Yaskawa INFORM job: OK_R2_O57-69(2)(90,0)_OK.JBI

/JOB
//NAME OK_R2_O57-69(2)(90,0)_OK
///FOLDERNAME X4
//POS
///NPOS 520,520,520,19,0,0
///TOOL 0
///POSTYPE PULSE
///PULSE
C00000=135424,72899,29147,3537,85342,-3792
C00001=134013,95021,61136,4029,77105,-4505
C00002=134047,101087,71818,4077,73656,-4607
C00003=134047,101216,72822,4088,73105,-4626
C00004=134047,101094,71866,4078,73630,-4609
C00005=133936,105187,77198,4137,72460,-4688
C00006=134047,101094,71866,4078,73630,-4609
C00007=133891,92563,58880,4064,77236,-4542
C00008=133627,85963,47659,4101,80754,-4516
C00009=133378,81291,43989,7801,81727,-8797
C00010=135556,84120,49328,8109,79955,-9206
C00011=135353,86004,57272,9537,76429,-10987
C00012=135353,86080,58384,9559,75792,-11036
C00013=135353,86004,57272,9537,76429,-10987
C00014=135153,91305,63913,9646,75106,-11159
C00015=135353,86004,57272,9537,76429,-10987
C00016=133639,82412,51163,9948,78523,-11411
C00017=132974,76709,41280,10049,81708,-11379
C00018=129415,64165,26444,10967,84795,-12306
C00019=98130,23251,42660,41088,49358,-30036
C00020=100023,30312,51600,41655,47069,-30160
C00021=100756,35138,59019,42789,45164,-30789
C00022=100756,36680,62008,43506,44389,-31244
C00023=100756,35138,59019,42789,45164,-30789
C00024=101219,36605,60555,42806,44807,-30721
C00025=100756,35138,59019,42789,45164,-30789
C00026=97195,22233,43091,41783,49188,-30648
C00027=75566,-7998,8685,42436,90764,-48719
C00028=92276,-23915,-5509,33057,78026,-45242
C00029=92276,-23145,-3597,33137,77364,-45439
C00030=92276,-23560,-4626,33093,77717,-45333
C00031=120131,-37031,-23614,-4680,71033,-34550
C00032=120131,-36585,-22326,-4696,70470,-34528
C00033=120989,-36588,-22328,-4847,70519,-34222
C00034=120131,-36585,-22326,-4696,70470,-34528
C00035=120131,-40902,-37029,-4549,77279,-34785
C00036=99101,-76935,-92016,31014,74911,-20401
C00037=52587,-144740,-101483,60524,64363,65274
C00038=46989,-65360,-59229,62781,73103,77672
C00039=56832,-65466,-56421,59287,64983,77772
C00040=57148,-65688,-55453,59188,64110,77279
C00041=55649,-62097,-53047,61106,66880,78547
C00042=57237,-59710,-51792,60669,66110,79037
C00043=56277,-61326,-53166,60831,66721,78866
C00044=55441,-62561,-53810,61057,67127,78609
C00045=56207,-63985,-54541,61032,66503,78630
C00046=55438,-62578,-53813,61060,67126,78606
C00047=51973,-62323,-54701,62406,69323,78001
C00048=48054,-62529,-57040,62601,72472,77896
C00049=29811,-70761,-60283,66780,94863,53671
C00050=30965,-22538,-31531,67696,97011,56857
C00051=55044,-42598,-44870,68563,88788,43678
C00052=56249,-45120,-46406,68472,87844,43687
C00053=57925,-45354,-44812,68371,86292,43442
C00054=57925,-45174,-43802,68390,86084,43215
C00055=57925,-45354,-44812,68371,86292,43442
C00056=59167,-45210,-44726,68282,85469,43617
C00057=57925,-45354,-44812,68371,86292,43442
C00058=55819,-44223,-45863,68504,88181,43684
C00059=44722,-31045,-43816,69927,97696,44632
C00060=43071,-26445,-40665,70170,98951,44614
C00061=137799,-47230,-78474,-21502,98719,52766
C00062=127020,6423,-39070,-7004,99714,51816
C00063=127020,5137,-37554,-6966,98131,51906
C00064=128416,4382,-35850,-7239,96821,52416
C00065=128416,3847,-35017,-7224,96041,52460
C00066=128416,4148,-35496,-7233,96488,52435
C00067=130041,4566,-35136,-7580,96617,52937
C00068=129924,4205,-34639,-7545,96120,52933
C00069=129457,4078,-34747,-7447,96082,52788
C00070=130190,4712,-35256,-7614,96778,52976
C00071=132441,34102,-13092,-8124,98426,53576
C00072=149392,-6912,-25974,-9982,75562,31317
C00073=149173,-488,-12666,-10148,70714,31647
C00074=149173,-326,-10897,-10208,69722,31733
C00075=149173,-394,-11578,-10184,70101,31701
C00076=148123,2416,-9216,-9823,69962,31333
C00077=149173,-394,-11578,-10184,70101,31701
C00078=152478,4885,-6741,-15795,72623,37698
C00079=151455,3828,-7649,-15488,72442,37350
C00080=152478,4560,-12614,-15554,75946,37261
C00081=146445,-24647,-43161,-13522,78564,34847
C00082=131494,-80468,-98534,-7816,92108,53678
C00083=52065,-14099,-27709,42253,108676,-27596
C00084=76671,-130461,-121705,35735,90710,-50834
C00085=94829,-93442,-100428,28991,96183,-47377
C00086=110716,-92055,-82664,19311,98038,-51285
C00087=114275,-93352,-80055,19461,95045,-50478
C00088=118122,-92212,-76367,19656,92534,-49497
C00089=118129,-91398,-74848,19645,92046,-49575
C00090=118122,-92212,-76367,19656,92534,-49497
C00091=119808,-92271,-76389,19753,92113,-48959
C00092=118122,-92212,-76367,19656,92534,-49497
C00093=114499,-91094,-78376,19482,95112,-50387
C00094=110992,-89821,-80983,19339,98080,-51178
C00095=124454,-89651,-86550,-11137,94998,69701
C00096=122569,-92184,-83910,-11067,91866,69331
C00097=120652,-93960,-80852,-11027,88857,68936
C00098=120652,-93520,-79457,-11027,88237,68992
C00099=120652,-93960,-80852,-11027,88857,68936
C00100=120650,-97396,-81866,-11026,87737,69033
C00101=120652,-93960,-80852,-11027,88857,68936
C00102=118161,-93768,-80427,-10994,88357,68121
C00103=120652,-93960,-80852,-11027,88857,68936
C00104=120037,-91891,-82714,-11032,90945,68539
C00105=121981,-89592,-85452,-11099,94026,68936
C00106=122005,-89480,-97857,-11363,101580,68254
C00107=122005,-89427,-98101,-11372,101754,68238
C00108=119094,-95812,-115555,4544,90851,20867
C00109=116502,-111480,-109655,18779,62868,-21987
C00110=119472,-101923,-104261,17094,63743,-20698
C00111=121534,-96097,-100090,16016,63743,-19914
C00112=121534,-96194,-98882,16123,62979,-20025
C00113=112336,-84014,-94514,26506,72534,-27449
C00114=114298,-84401,-94682,25743,71847,-26864
C00115=121534,-96097,-100090,16016,63743,-19914
C00116=121514,-92242,-98700,15883,64832,-19765
C00117=121534,-96097,-100090,16016,63743,-19914
C00118=119823,-101836,-103002,17025,62972,-20682
C00119=116876,-111303,-108368,18711,62117,-21969
C00120=126032,-109701,-108999,-21760,66785,27050
C00121=122513,-101468,-103921,-20079,66940,25677
C00122=121483,-94377,-99419,-19507,67520,25186
C00123=121483,-94509,-98158,-19621,66724,25324
C00124=121483,-94377,-99419,-19507,67520,25186
C00125=119206,-94355,-99408,-18489,67008,24418
C00126=121483,-94377,-99419,-19507,67520,25186
C00127=121468,-91005,-98354,-19362,68535,25006
C00128=121483,-94377,-99419,-19507,67520,25186
C00129=124810,-108862,-107603,-21303,66070,26716
C00130=126981,-112864,-109311,-24940,61360,29729
C00131=123200,-104180,-104415,-22777,61614,28126
C00132=121230,-90686,-98732,-21152,64298,26805
C00133=121230,-90968,-97120,-21351,63235,27013
C00134=121230,-90806,-98119,-21226,63888,26884
C00135=118688,-90754,-98099,-19926,63280,26013
C00136=121230,-90721,-98563,-21173,64184,26826
C00137=121211,-84894,-96124,-20922,65577,26553
C00138=121230,-90686,-98732,-21152,64298,26805
C00139=121413,-93580,-100796,-21282,64141,26906
C00140=124847,-101623,-105736,-23178,64029,28268
C00141=120616,-95755,-103879,-23668,64726,45447
C00142=120621,-89459,-99052,-23623,64971,45396
C00143=103351,-79665,-99305,-783,71297,41010
C00144=120614,-97387,-102466,-23992,63157,45792
C00145=122354,-96256,-100860,-24938,63287,46459
C00146=100033,-102933,-105835,1367,63570,39915
C00147=94055,-138721,-112948,5183,49813,37109
C00148=86627,-164185,-115821,11591,39368,32593
C00149=96470,-180165,-126119,4784,36529,37522
C00150=120616,-95173,-105764,-23303,89544,42444
C00151=107191,-96001,-89285,-21702,28532,58770
C00152=107187,-93630,-79997,-25295,24388,60561
C00153=107188,-92928,-77886,-26213,23539,61010
C00154=112799,-77365,-77001,-28703,40381,63534
C00155=107081,-94020,-78768,-26067,23489,60939
C00156=108911,-93070,-77209,-29349,23678,62538
C00157=100995,-91828,-91259,-7616,48178,54187
C00158=103021,-103152,-96284,-14725,52035,64235
C00159=107822,-73722,-90278,-18203,77746,63273
C00160=110657,-50226,-86705,-20295,96355,61815
C00161=107202,-93991,-108886,-21178,109925,43661
C00162=120660,-73953,-111348,-177,99224,-835
C00163=120616,-96234,-101081,23944,56754,-46777
C00164=120615,-96493,-97034,24670,54353,-47364
C00165=120614,-96447,-94923,25055,53191,-47662
C00166=125103,-63544,-87949,17256,75790,-41512
C00167=118876,-96360,-94049,26267,53277,-48431
C00168=120612,-97621,-95709,25094,53083,-47691
C00169=123782,-105215,-109377,22364,82684,-38148
C00170=123367,-104493,-108204,22899,85714,-42144
C00171=120617,-94319,-107453,23464,90858,-42123
C00172=120617,-92878,-109780,23521,92858,-41729
C00173=120619,-86141,-115603,23930,99335,-40429
C00174=120619,-89012,-115558,-8782,73464,-77384
C00175=120618,-92353,-112869,-8941,70132,-77138
C00176=120618,-93422,-111698,-9011,68877,-77043
C00177=120616,-94109,-113157,-8979,69414,-77085
C00178=120318,-89311,-110489,-8778,70198,-77244
C00179=120618,-93688,-111329,-9132,68044,-76969
C00180=120618,-93957,-110924,-9216,67187,-76884
C00181=120618,-94299,-110440,-9161,65769,-76809
C00182=120618,-94831,-109599,-8469,63241,-76696
C00183=120617,-95145,-109027,-7071,61401,-76664
C00184=120617,-95217,-108863,-5672,60665,-76701
C00185=120618,-93036,-111930,-4923,63538,-76718
C00186=120618,-92960,-112001,-4009,63579,-76743
C00187=120618,-92691,-112274,-2433,64167,-76800
C00188=120618,-92166,-112798,-840,65602,-76863
C00189=120618,-91419,-113490,342,67708,-76910
C00190=120619,-90739,-114068,878,69589,-76936
C00191=120619,-89701,-115007,939,71612,-76812
C00192=120619,-88814,-115609,873,73870,-76855
C00193=120619,-87740,-116270,151,76574,-76959
C00194=120619,-86987,-116700,-1182,78540,-77121
C00195=120619,-86782,-116823,-2462,79296,-77267
C00196=120619,-90672,-114378,-3278,75949,-77117
C00197=120619,-90769,-114313,-4130,75889,-77177
C00198=120619,-91109,-114056,-5597,75252,-77256
C00199=120618,-91719,-113544,-7101,73764,-77286
C00200=120618,-92472,-112836,-8259,71637,-77242
C00201=120618,-92872,-112418,-8666,70405,-77193
C00202=120618,-93168,-112034,-8862,69621,-77111
C00203=120618,-93422,-111698,-9011,68877,-77043
C00204=120618,-92353,-112869,-8941,70132,-77138
C00205=120619,-89012,-115558,-8782,73464,-77384
C00206=120595,-119438,-127420,8829,91162,-8830
C00207=129025,-103888,-99333,-21372,86937,54976
C00208=120613,-94952,-86848,-20336,81911,52813
C00209=120613,-94069,-83278,-20415,80272,53091
C00210=106776,-118156,-87795,-9907,57184,33367
C00211=120519,-95091,-83551,-20421,79912,53118
C00212=122104,-92396,-81537,-20633,80446,53604
C00213=112247,-111724,-87315,-12944,66201,41339
C00214=120203,-93448,-81675,-16163,85448,56808
C00215=120729,-92509,-78586,-16225,84191,57156
C00216=121550,-94129,-79175,-15118,86186,61621
C00217=122418,-96212,-79737,-13214,89323,68733
C00218=120612,-93818,-82398,-13271,91824,67835
C00219=120613,-94827,-86367,-13308,93699,67633
C00220=120614,-96085,-95173,-13466,98348,67128
C00221=120625,-105302,-100360,-13404,96846,67297
C00222=102872,-120945,-93289,41313,52454,-35552
C00223=111052,-89986,-73102,36259,51528,-31574
C00224=114360,-89865,-71590,35102,49434,-30694
C00225=117526,-83033,-67896,32906,49195,-29120
C00226=113966,-89555,-70876,35431,49366,-30932
C00227=115650,-91167,-72721,34446,48930,-30213
C00228=116035,-87162,-73783,30522,57415,-33049
C00229=114870,-90750,-79036,28299,65889,-37708
C00230=114629,-93248,-83330,25887,75293,-43435
C00231=115086,-85156,-72081,25020,76812,-47005
C00232=114845,-96650,-75395,24460,77575,-52847
C00233=115266,-96292,-75579,23738,83016,-58597
C00234=112822,-91718,-77371,23458,91001,-62960
C00235=109330,-92095,-80656,23399,93677,-63722
C00236=110759,-94815,-97268,24043,101385,-61640
C00237=25230,-87703,-86789,41333,106155,71905
C00238=55862,19660,17206,68346,89547,53836
C00239=59225,37567,25812,69215,105770,42705
C00240=67658,42850,42597,68102,97125,40508
C00241=69496,40939,42743,68154,95469,40297
C00242=67599,42910,43858,67984,96867,40179
C00243=68366,42138,41747,68199,96713,40671
C00244=69496,40844,42642,68155,95474,40303
C00245=69202,26042,27763,68892,91580,41859
C00246=69430,8343,11443,69273,87154,43187
C00247=70515,-11168,-4593,69437,78895,44683
C00248=70497,-3239,1595,68550,83825,57162
C00249=68177,-4212,-1280,68454,85880,57398
C00250=65815,-3605,-3490,68417,88124,57797
C00251=46513,-27715,-22241,69125,80479,38621
C00252=7625,-19791,-74194,84461,116832,51132
C00253=98528,-26744,-48644,33463,55012,18344
C00254=113253,15209,27106,3834,50657,-3406
C00255=113409,21623,32322,3755,50736,-3338
C00256=112944,26693,40965,4138,48051,-3650
C00257=113472,24070,39362,3899,47665,-3430
C00258=113579,25546,39455,3805,48359,-3355
C00259=112978,26683,40955,4121,48050,-3635
C00260=112942,28151,43799,5754,47269,-5081
C00261=107858,34053,50994,19891,49698,-15260
C00262=107375,37871,55183,23682,51778,-19403
C00263=102416,58013,78822,34430,58031,-35011
C00264=101528,71839,96969,38749,59697,-40411
C00265=101833,70144,94845,38592,59915,-40184
C00266=99205,63215,84174,37575,62603,-39615
C00267=97180,56339,73463,36771,65900,-39269
C00268=108272,10166,23438,3323,45242,-19316
C00269=109103,10218,12469,2549,51979,-18742
C00270=102461,24196,25876,17974,57306,-30655
C00271=99785,30090,30578,21838,60128,-34061
C00272=99052,29053,30612,22206,59809,-34434
C00273=101478,26267,28203,21358,59216,-33547
C00274=98901,31355,34377,29186,63057,-41116
C00275=92009,66840,89116,42947,61850,-57046
C00276=89877,62120,80876,42077,64804,-56709
C00277=70258,15873,38394,48666,102593,-69187
C00278=68720,8010,42290,53616,94090,-68666
C00279=74407,27282,60534,55400,90233,-68095
C00280=74758,1474,21309,45746,90270,-65676
C00281=98607,12568,39814,-52966,86937,-78252
C00282=98596,22842,59344,-53301,82774,-75788
C00283=96296,21421,60413,-54092,80731,-75703
C00284=95348,20952,60953,-54433,79893,-75663
C00285=96117,19164,58324,-54129,80713,-75783
C00286=95662,23434,63388,-54370,79922,-75521
C00287=95503,21312,61702,-54422,79811,-75531
C00288=92574,18445,54645,-48983,79889,-68258
C00289=91800,17848,53101,-47601,79897,-67557
C00290=92530,17999,51917,-47342,80806,-67673
C00291=94302,18640,49262,-46764,83033,-67943
C00292=79003,18324,29303,-31626,94586,-4503
C00293=64136,40618,57122,-29721,84915,-83830
C00294=62802,39067,58740,-29997,82892,-83805
C00295=62255,38544,59506,-30121,82059,-83791
C00296=62254,37103,56589,-30066,82978,-84033
C00297=62821,40643,61741,-30049,81995,-83562
C00298=59984,48909,70165,-26795,84201,-83115
C00299=59410,69261,96131,-25367,86084,-74959
C00300=59404,69357,96256,-25356,86081,-74939
C00301=59713,70793,96681,-25260,86600,-74945
C00302=60461,74839,98386,-25037,87745,-74932
C00303=60470,59585,70460,-25309,96249,-76737
C00304=66845,10330,41939,-25249,64720,-33768
C00305=66816,16396,52426,-25952,61688,-33052
C00306=66804,19142,57057,-26292,60387,-32730
C00307=66058,20615,58344,-26298,60142,-32956
C00308=66868,17219,53699,-26035,61378,-32955
C00309=66973,19658,57552,-26302,60399,-32669
C00310=66985,16895,52895,-25961,61707,-32992
C00311=67015,10800,42362,-25255,64752,-33711
C00312=98181,31350,57269,-53093,86032,-77938
C00313=96082,29267,57446,-53647,84171,-77916
C00314=95219,28523,57622,-53885,83405,-77901
C00315=95917,26905,55160,-53675,84199,-78019
C00316=95506,31088,60230,-53837,83386,-77740
C00317=95359,28788,58259,-53869,83329,-77779
C00318=92697,26913,52373,-48450,83827,-70215
C00319=91994,26523,51069,-47073,83939,-69440
C00320=92656,26997,50292,-46905,84772,-69532
C00321=94270,28412,48618,-46533,86809,-69749
C00322=79891,40483,43632,-25605,98381,17488
C00323=64421,55368,61348,-15926,95442,62339
C00324=63205,52871,61672,-16144,93779,62133
C00325=62708,51961,61917,-16235,93087,62052
C00326=62707,50761,59239,-16263,94078,61920
C00327=63223,54241,64482,-16113,92796,62269
C00328=60236,62044,73663,-12795,94061,63101
C00329=59090,69141,83012,-10500,94867,70833
C00330=59083,69182,83067,-10487,94869,70851
C00331=59379,71028,84054,-10408,95242,70919
C00332=60098,76023,87068,-10213,96031,71094
C00333=60107,66003,66038,-10511,103704,70448
C00334=66860,35146,61423,-22993,49349,-53528
C00335=66834,42827,74568,-24499,45535,-52525
C00336=66824,46660,80883,-25305,43786,-52015
C00337=66175,48781,83167,-25255,43321,-52183
C00338=66880,43946,76304,-24713,45097,-52378
C00339=66970,47398,81721,-25407,43702,-51920
C00340=66981,43500,75311,-24586,45473,-52438
C00341=67007,35727,62031,-23060,49318,-53454
C00342=87565,40229,55167,-37616,76398,-68031
C00343=104252,61764,84947,-51561,88394,-76219
C00344=102517,58043,82852,-52038,87086,-76344
C00345=101804,56689,82195,-52237,86527,-76380
C00346=102435,54601,78919,-52052,87454,-76595
C00347=101993,60636,86873,-52209,86091,-76036
C00348=101932,57147,83104,-52210,86393,-76238
C00349=99529,53434,74771,-46937,87155,-68655
C00350=98895,52660,72970,-45595,87312,-67859
C00351=99433,53501,72680,-45467,88010,-67934
C00352=100745,55861,72292,-45181,89689,-68100
C00353=89942,52639,54543,-22757,100290,22350
C00354=84530,60242,66965,-10989,97828,69052
C00355=83700,56528,65849,-11170,96516,68885
C00356=83359,55133,65530,-11245,95959,68819
C00357=83358,53843,62725,-11276,97003,68723
C00358=83705,58033,68848,-11139,95464,68982
C00359=80399,62193,73871,-7256,96460,69699
C00360=78998,67441,80988,-4366,97017,77318
C00361=78990,67470,81028,-4351,97018,77335
C00362=79114,69587,82331,-4315,97310,77366
C00363=79414,75293,86196,-4226,97877,77446
C00364=79422,65472,65446,-4368,105580,77179
C00365=80352,27457,54566,-26195,53383,-48637
C00366=80356,27473,54581,-26196,53382,-48635
C00367=80357,27479,54587,-26196,53382,-48634
C00368=79589,28666,55655,-26054,53112,-48894
C00369=80424,25883,51570,-25884,54338,-48863
C00370=80357,27479,54587,-26196,53382,-48634
C00371=80356,27473,54581,-26196,53382,-48635
C00372=80352,27458,54566,-26195,53383,-48637
C00373=110061,-17560,-36552,-26636,92274,-45980
C00374=111839,-83491,-103870,-27371,99587,-47031
C00375=38426,-40229,-52385,46753,77455,20722
C00376=20805,-37224,-43776,64442,70782,24410
C00377=53615,-60479,-29767,71413,48188,35364
C00378=53622,-60473,-29764,71411,48184,35366
C00379=53625,-60471,-29763,71411,48182,35366
C00380=52450,-61746,-30400,71683,48877,35041
C00381=53622,-61330,-31549,70858,48414,35743
C00382=53667,-60425,-29740,73440,59962,39458
C00383=53705,-60384,-29719,74506,70698,55233
C00384=53706,-60382,-29718,74560,71274,55582
C00385=53707,-60381,-29717,74560,71274,55582
C00386=53710,-60377,-29715,74560,71273,55583
C00387=53701,-60384,-29719,74560,71278,55581
C00388=66706,-54450,-33709,25643,46200,1067
C00389=66709,-54445,-33707,25641,46199,1069
C00390=65806,-56035,-34565,26242,46218,617
C00391=67582,-55929,-35261,25089,46110,1484
C00392=66709,-54446,-33707,25645,46199,1067
C00393=66709,-54446,-33707,25645,46199,1067
C00394=66709,-54447,-33708,25641,46199,1069
C00395=66706,-54452,-33711,25643,46199,1067
C00396=56114,-41526,-33189,36880,64877,-1074
C00397=62492,-26274,-11536,67617,51989,49416
C00398=67015,-30786,-7269,70211,42036,48662
C00399=67021,-30777,-7263,70209,42033,48664
C00400=67024,-30773,-7260,70208,42031,48665
C00401=67025,-30771,-7259,70208,42030,48665
C00402=66245,-32305,-8266,70488,42489,48421
C00403=67024,-31573,-9128,69442,42305,49131
C00404=67037,-30747,-7244,72021,47713,46269
C00405=67060,-30703,-7215,71923,58333,61620
C00406=67063,-30697,-7211,72128,59825,62445
C00407=67063,-30696,-7209,72128,59824,62445
C00408=67065,-30691,-7207,72128,59824,62445
C00409=67053,-30709,-7218,72128,59831,62443
C00410=67069,40537,9457,57195,76262,35492
C00411=67067,40166,11985,57536,75289,34802
C00412=67066,40064,13042,57682,74899,34523
C00413=66577,38326,11242,57768,75308,34517
C00414=67065,40169,11907,57527,75318,34822
C00415=67072,40075,13170,59772,79795,32172
C00416=67078,40614,25191,75815,82535,42307
C00417=67079,40861,26780,77445,83659,42995
C00418=67080,40685,25622,77394,83811,43275
C00419=67085,40340,22831,77277,84191,43970
C00420=67090,40073,14255,76963,85485,46282
C00421=90837,-14160,-23602,46112,79870,-29092
C00422=94881,-86110,-91503,45134,79065,-22948
C00423=94881,-86110,-91503,45134,79065,-22948
C00424=94881,-86110,-91503,45134,79065,-22948
C00425=64023,-117945,-92652,70836,68337,59810
C00426=77839,-63283,-64145,64455,63318,66711
C00427=80052,-65654,-65354,64094,61673,66872
C00428=91733,-74743,-69530,58015,49641,61106
C00429=80955,-66618,-66084,63874,61070,67008
C00430=80000,-68279,-65664,64663,61180,66324
C00431=91573,-74565,-69447,58050,49760,61088
C00432=100815,-86079,-74448,43553,32020,68906
C00433=93567,-76904,-70333,47145,37282,67091
C00434=87612,-64523,-64419,48752,42307,66391
C00435=94575,-77342,-71004,49651,37504,40583
C00436=95005,-77606,-71124,49413,37228,40705
C00437=25543,-37396,-56331,69239,85891,31897
C00438=172418,-62024,-69195,-63943,69139,-25706
C00439=192822,-61773,-75094,-68063,83874,-24345
C00440=147462,40071,30365,-69170,75532,-19593
C00441=147457,40119,30415,-69171,75526,-19591
C00442=147456,40127,30423,-69171,75525,-19590
C00443=147721,37841,28052,-69134,75813,-19681
C00444=148042,40615,30212,-69143,76066,-19681
C00445=147457,40126,30423,-69172,75522,-19590
C00446=147457,40126,30423,-69172,75522,-19590
C00447=147457,40125,30422,-69171,75526,-19590
C00448=147458,40117,30413,-69171,75527,-19591
C00449=147460,40097,30392,-69171,75529,-19592
C00450=134071,6209,-12454,-63265,71876,-23505
C00451=134070,6228,-12438,-63265,71875,-23505
C00452=134070,6235,-12431,-63265,71875,-23505
C00453=134229,4110,-14261,-63296,71992,-23494
C00454=134787,6570,-12855,-63330,72532,-23573
C00455=134070,6235,-12432,-63265,71872,-23505
C00456=134070,6235,-12432,-63265,71872,-23505
C00457=134071,6233,-12433,-63265,71876,-23505
C00458=134071,6226,-12439,-63265,71876,-23505
C00459=134072,6208,-12455,-63265,71877,-23505
C00460=134072,6180,-12479,-63265,71877,-23505
C00461=130462,-25122,-37090,-45275,45470,-33351
C00462=132886,-107940,-72929,-67003,34868,-20711
C00463=175339,-34674,-82182,-59494,83195,-32396
C00464=136096,14126,-32620,-12825,85534,-21552
C00465=129268,64776,27312,8163,83182,-8944
C00466=134681,94635,47335,809,84864,-881
C00467=133307,94687,54997,-6000,80862,2911
C00468=132876,99561,59391,7151,80998,-7884
C00469=132758,96232,56359,7183,81163,-7913
C00470=134709,101130,63695,-5988,78818,2671
C00471=135101,106095,70233,-5013,77180,1553
C00472=133232,101987,65437,-241,76556,-4364
C00473=130942,105736,66959,6239,79029,-10361
C00474=131542,110305,67283,11855,83586,-13328
C00475=129370,129654,73054,9751,92339,-13599
C00476=127763,125744,69167,15594,92406,-13107
C00477=127928,126623,70430,17139,93326,-15161
C00478=128241,125871,69474,17076,93457,-15039
C00479=129815,119231,60338,14426,93579,-11375
C00480=130278,118783,59618,14311,93713,-11211
C00481=129188,114780,51212,14689,96908,-11178
C00482=127389,122324,63446,15731,94168,-13005
C00483=137764,36598,17142,-9265,69493,-22853
C00484=175415,-48371,-56760,-63540,71824,-23104
C00485=132886,-114094,-83669,-62634,36414,-23122
C00486=105972,-102146,-97903,-7412,79578,37972
C00487=160165,-110950,-92023,-21545,85745,61448
C00488=140609,-94579,-78221,-8463,77656,55534
C00489=138726,-94535,-76086,-8242,76183,54976
C00490=163390,-101496,-77356,-21709,82707,63168
C00491=161792,-103413,-79036,-21690,82331,62654
C00492=135933,-74368,-67331,-7717,80836,53706
C00493=133468,-45426,-54020,-7292,87230,52484
C00494=132807,-44691,-51453,-7196,85977,52334
C00495=131271,-21709,-36375,-6964,88353,51682
C00496=131369,-18521,-50976,-7106,98910,51122
C00497=155973,17568,-14616,-23088,90451,45565
C00498=155497,22906,-1419,-24756,87977,49189
C00499=156165,24198,2743,-24323,85495,48766
C00500=157855,17140,-6636,-24602,87944,48876
C00501=148516,-1587,-23042,-9652,76377,30951
C00502=147710,1301,-17894,-9446,74621,30813
C00503=138722,3472,-16218,8570,74426,13517
C00504=137116,-4059,-28477,8993,78231,13244
C00505=138249,-10506,-39760,1549,83744,18421
C00506=145553,-65590,-46111,-45971,69798,51566
C00507=117087,2274,-4333,74835,51753,-34811
C00508=120822,45639,36263,74296,46580,-35142
C00509=132292,76688,41038,57812,44611,-25328
C00510=133587,85399,43635,54635,45518,-23471
C00511=134089,87151,52872,58446,42500,-25922
C00512=133465,87868,53767,58981,42776,-26187
C00513=134426,84651,49764,57666,42643,-25479
C00514=134089,87030,55209,59870,41700,-26787
C00515=134090,96417,89471,79265,35490,-37858
C00516=134090,100042,96821,83028,34997,-39924
C00517=133589,94413,89775,81024,35602,-38850
C00518=132294,83338,76456,77824,37058,-37121
C00519=-3643,-66769,-111182,-19341,79018,-78067
BC00000=138390,352725,245958
BC00001=138390,352725,245958
BC00002=138390,352725,245958
BC00003=138390,352725,245958
BC00004=138390,352725,245958
BC00005=138390,352725,245958
BC00006=138390,352725,245958
BC00007=138390,352725,245958
BC00008=138390,352725,245958
BC00009=131940,350742,262337
BC00010=129582,350248,253511
BC00011=128096,349560,276971
BC00012=128096,349560,276971
BC00013=128096,349560,276971
BC00014=128096,349560,276971
BC00015=128096,349560,276971
BC00016=128096,349560,276971
BC00017=128096,349560,276971
BC00018=128096,349560,276971
BC00019=111959,352484,367172
BC00020=111959,352484,367172
BC00021=111959,352484,367172
BC00022=111959,352484,367172
BC00023=111959,352484,367172
BC00024=111960,352483,367169
BC00025=111959,352484,367172
BC00026=111959,352484,367172
BC00027=111959,352484,367172
BC00028=111959,352484,367172
BC00029=111959,352484,367172
BC00030=111959,352484,367172
BC00031=111959,352484,367172
BC00032=111959,352484,367172
BC00033=111959,352484,367172
BC00034=111959,352484,367172
BC00035=111959,352484,367172
BC00036=111562,519678,418259
BC00037=342634,456988,86611
BC00038=339612,461620,87060
BC00039=339612,461620,87060
BC00040=339612,461620,87060
BC00041=339612,461620,87060
BC00042=339612,461620,87060
BC00043=339612,461620,87060
BC00044=339612,461620,87060
BC00045=339612,461620,87060
BC00046=339612,461620,87060
BC00047=339612,461620,87060
BC00048=339612,461620,87060
BC00049=369424,454605,90098
BC00050=369424,454605,90098
BC00051=398158,448947,97388
BC00052=398158,444723,78431
BC00053=398158,443034,70848
BC00054=398158,443034,70848
BC00055=398158,443034,70848
BC00056=398158,443034,70848
BC00057=398158,443034,70848
BC00058=398158,445606,70943
BC00059=398158,449830,89900
BC00060=398158,496460,89900
BC00061=309723,504773,89900
BC00062=309723,472531,89900
BC00063=309723,472531,89900
BC00064=309723,472531,89900
BC00065=309723,472531,89900
BC00066=309723,472531,89900
BC00067=309723,472531,89900
BC00068=309723,472531,89900
BC00069=309723,472531,89900
BC00070=309723,472531,89900
BC00071=309723,472531,89900
BC00072=311190,379628,212757
BC00073=311190,379628,212757
BC00074=311190,379628,212757
BC00075=311190,379628,212757
BC00076=311190,379628,212757
BC00077=311190,379628,212757
BC00078=311190,379628,212757
BC00079=311190,379628,212757
BC00080=311190,379628,212757
BC00081=311190,379628,212757
BC00082=309723,472531,89900
BC00083=302213,518265,714952
BC00084=365185,474930,1004970
BC00085=376205,445622,992724
BC00086=398158,419651,1075139
BC00087=398158,419651,1075139
BC00088=398158,419651,1075139
BC00089=398158,419651,1075139
BC00090=398158,419651,1075139
BC00091=398158,419651,1075139
BC00092=398158,419651,1075139
BC00093=398158,419651,1075139
BC00094=398158,419651,1075139
BC00095=395948,423266,1075139
BC00096=395948,423266,1075139
BC00097=395948,423266,1075139
BC00098=395948,423266,1075139
BC00099=395948,423266,1075139
BC00100=395948,423266,1075139
BC00101=395948,423266,1075139
BC00102=395948,423266,1075139
BC00103=395948,423266,1075139
BC00104=395948,423266,1075139
BC00105=395948,423266,1075139
BC00106=395948,423266,1075139
BC00107=395948,423266,1075139
BC00108=340598,374601,1075139
BC00109=291299,331257,1075139
BC00110=291299,331257,1075139
BC00111=291299,331257,1075139
BC00112=291299,331257,1075139
BC00113=291298,331257,1075136
BC00114=291299,331257,1075139
BC00115=291299,331257,1075139
BC00116=291299,331257,1075139
BC00117=291299,331257,1075139
BC00118=291299,331257,1075139
BC00119=291299,331257,1075139
BC00120=261372,332564,1075139
BC00121=261372,332564,1075139
BC00122=261372,332564,1075139
BC00123=261372,332564,1075139
BC00124=261372,332564,1075139
BC00125=261372,332564,1075139
BC00126=261372,332564,1075139
BC00127=261372,332564,1075139
BC00128=261372,332564,1075139
BC00129=261372,332564,1075139
BC00130=307746,348207,1075139
BC00131=307746,348207,1075139
BC00132=307746,348207,1075139
BC00133=307746,348207,1075139
BC00134=307746,348207,1075139
BC00135=307746,348207,1075139
BC00136=307746,348207,1075139
BC00137=307746,348207,1075139
BC00138=307746,348207,1075139
BC00139=307746,348207,1075139
BC00140=307746,348207,1075139
BC00141=295789,345827,1075139
BC00142=301228,342160,1075139
BC00143=301229,342159,1075135
BC00144=303404,340694,1075139
BC00145=303404,340694,1075139
BC00146=301229,342159,1075135
BC00147=301229,342159,1075135
BC00148=301229,342159,1075135
BC00149=301229,342159,1075135
BC00150=292398,348738,1075139
BC00151=232590,368151,1075139
BC00152=232611,368148,1075139
BC00153=237632,363214,1075139
BC00154=239639,361241,1075138
BC00155=239640,361241,1075139
BC00156=239640,361241,1075139
BC00157=236201,347334,1075139
BC00158=236201,347334,1075139
BC00159=236201,347334,1075139
BC00160=236201,347334,1075139
BC00161=235432,272930,1075139
BC00162=281159,319039,1075139
BC00163=310685,343195,1075139
BC00164=310695,343194,1075139
BC00165=305405,338959,1075139
BC00166=305405,338959,1075139
BC00167=303288,337266,1075139
BC00168=303288,337266,1075139
BC00169=309165,291369,1075139
BC00170=309175,293011,1075139
BC00171=311437,296205,1075139
BC00172=317053,297452,1075139
BC00173=317032,297454,1075139
BC00174=38645,323428,1075139
BC00175=39322,320899,1075139
BC00176=39592,319888,1075139
BC00177=39592,319888,1075139
BC00178=39592,319888,1075139
BC00179=44164,321385,1075139
BC00180=49926,323066,1075139
BC00181=50935,324538,1075139
BC00182=53180,326990,1075139
BC00183=56412,328576,1075139
BC00184=59240,328893,1075139
BC00185=64280,309350,1075139
BC00186=65993,309027,1075139
BC00187=68725,308060,1075139
BC00188=71288,306312,1075139
BC00189=72971,303977,1075139
BC00190=73362,301969,1075139
BC00191=51582,297025,1075139
BC00192=50713,294790,1075139
BC00193=48610,292273,1075139
BC00194=45444,290610,1075139
BC00195=42623,290262,1075139
BC00196=37229,309748,1075139
BC00197=35508,310080,1075139
BC00198=32776,311095,1075139
BC00199=30259,312932,1075139
BC00200=28686,315356,1075139
BC00201=28637,316774,1075139
BC00202=35085,318487,1075139
BC00203=39592,319888,1075139
BC00204=39322,320899,1075139
BC00205=38645,323428,1075139
BC00206=340546,340147,1075139
BC00207=386053,422772,1075139
BC00208=386053,422772,1075139
BC00209=391117,422740,1075139
BC00210=393141,422728,1075125
BC00211=393142,422726,1075139
BC00212=393142,422726,1075139
BC00213=394689,420137,1075130
BC00214=398158,414330,1075139
BC00215=389899,428595,1075139
BC00216=392082,424794,1075135
BC00217=395622,418632,1075139
BC00218=394381,417581,1075139
BC00219=391277,414954,1075139
BC00220=391256,414957,1075139
BC00221=391256,414957,1075139
BC00222=398158,443815,1075139
BC00223=398158,443813,1075139
BC00224=398158,438136,1075139
BC00225=398158,435866,1075139
BC00226=398158,435866,1075139
BC00227=398158,435866,1075139
BC00228=398158,426010,1075139
BC00229=398158,415040,1075139
BC00230=398158,401708,1075139
BC00231=398158,445460,1075139
BC00232=398158,437775,1075139
BC00233=398158,428690,1075139
BC00234=398158,421387,1075139
BC00235=398158,419412,1075139
BC00236=398158,423088,1075139
BC00237=305810,516728,1075139
BC00238=398158,495883,160317
BC00239=398158,479397,168150
BC00240=398158,479397,168150
BC00241=398158,479397,168150
BC00242=398158,479397,168150
BC00243=398158,479397,168150
BC00244=398158,479397,168150
BC00245=398158,479397,168150
BC00246=398158,479397,168150
BC00247=398158,479397,168150
BC00248=398158,479397,168150
BC00249=398158,479397,168150
BC00250=398158,479397,168150
BC00251=398158,495883,160317
BC00252=7949,495883,160317
BC00253=88409,416618,458299
BC00254=112807,351372,371410
BC00255=112807,351372,347240
BC00256=112807,351372,359623
BC00257=112807,351372,371410
BC00258=112807,351372,371410
BC00259=112807,351372,359623
BC00260=112807,351372,367422
BC00261=112807,351372,371410
BC00262=112807,351372,371410
BC00263=112807,351372,371410
BC00264=112807,351372,371410
BC00265=112807,351372,371410
BC00266=112807,351372,371410
BC00267=112807,351372,371410
BC00268=95901,348186,362946
BC00269=95901,348186,278544
BC00270=95902,348187,278542
BC00271=95902,348186,278541
BC00272=95902,348186,278541
BC00273=95902,348186,278541
BC00274=95902,348186,278544
BC00275=95901,348186,362946
BC00276=95901,348186,362946
BC00277=95901,348186,362946
BC00278=95901,348186,362946
BC00279=95901,348186,362946
BC00280=95901,348186,362946
BC00281=113744,387382,443450
BC00282=113744,387382,443450
BC00283=113744,387382,443450
BC00284=113744,387382,443450
BC00285=113744,387382,443450
BC00286=113744,387382,443450
BC00287=113744,387382,443450
BC00288=113744,387382,443450
BC00289=113744,387382,443450
BC00290=113744,387382,443450
BC00291=113744,387382,443450
BC00292=105209,380725,420258
BC00293=71135,367650,422598
BC00294=71135,367650,422598
BC00295=71135,367650,422598
BC00296=71135,367650,422598
BC00297=71135,367650,422598
BC00298=71135,367650,422598
BC00299=71135,367650,422598
BC00300=71135,367650,422598
BC00301=71135,367650,422598
BC00302=71135,367650,422598
BC00303=71135,367650,422598
BC00304=83700,393879,577285
BC00305=83700,393879,577285
BC00306=83700,393879,577285
BC00307=83700,393879,577285
BC00308=83700,393879,577285
BC00309=83700,393879,577285
BC00310=83700,393879,577285
BC00311=83700,393879,577285
BC00312=107452,368535,386004
BC00313=107452,368535,386004
BC00314=107452,368535,386004
BC00315=107452,368535,386004
BC00316=107452,368535,386004
BC00317=107452,368535,386004
BC00318=107452,368535,386004
BC00319=107452,368535,386004
BC00320=107452,368535,386004
BC00321=107452,368535,386004
BC00322=98501,369108,368404
BC00323=79824,352117,369823
BC00324=79824,352117,369823
BC00325=79824,352117,369823
BC00326=79824,352117,369823
BC00327=79824,352117,369823
BC00328=79824,352117,369823
BC00329=79824,352117,369823
BC00330=79824,352117,369823
BC00331=79824,352117,369823
BC00332=79824,352117,369823
BC00333=79824,352117,369823
BC00334=56231,402325,530501
BC00335=56231,402325,530501
BC00336=56231,402325,530501
BC00337=56231,402325,530501
BC00338=56231,402325,530501
BC00339=56231,402325,530501
BC00340=56231,402325,530501
BC00341=56231,402325,530501
BC00342=90082,380846,432093
BC00343=117586,363395,352136
BC00344=117586,363395,352136
BC00345=117586,363395,352136
BC00346=117586,363395,352136
BC00347=117586,363395,352136
BC00348=117586,363395,352136
BC00349=117586,363395,352136
BC00350=117586,363395,352136
BC00351=117586,363395,352136
BC00352=117586,363395,352136
BC00353=126861,357458,364185
BC00354=131499,354490,370210
BC00355=131499,354490,370210
BC00356=131499,354490,370210
BC00357=131499,354490,370210
BC00358=131499,354490,370210
BC00359=131499,354490,370210
BC00360=131499,354490,370210
BC00361=131499,354490,370210
BC00362=131499,354490,370210
BC00363=131499,354490,370210
BC00364=131499,354490,370210
BC00365=90764,380680,536482
BC00366=91452,379989,509808
BC00367=91727,379713,499139
BC00368=91727,379713,499139
BC00369=91727,379713,499139
BC00370=91729,379098,499145
BC00371=91454,379375,509815
BC00372=90766,380066,536489
BC00373=90764,380680,536482
BC00374=90764,512522,536482
BC00375=122162,478683,262546
BC00376=129550,465631,198091
BC00377=152465,451599,229687
BC00378=153172,446174,210806
BC00379=153455,444004,203254
BC00380=153455,444004,203254
BC00381=153455,444004,203254
BC00382=178403,442366,194004
BC00383=198722,435310,174556
BC00384=199688,434852,173431
BC00385=201465,436663,179712
BC00386=205908,441191,195414
BC00387=205898,441193,222298
BC00388=140845,446445,275017
BC00389=142184,444126,269603
BC00390=142184,444126,269603
BC00391=142184,444126,269603
BC00392=141310,444124,265365
BC00393=139445,444111,256387
BC00394=138563,444101,252166
BC00395=137223,446420,257580
BC00396=140845,446445,275017
BC00397=158126,451813,276188
BC00398=157660,453937,283582
BC00399=157670,453936,256698
BC00400=156850,448515,237853
BC00401=156522,446347,230315
BC00402=156522,446347,230315
BC00403=156522,446347,230315
BC00404=167171,445462,226404
BC00405=187235,438429,220120
BC00406=189797,437317,218030
BC00407=191574,439128,224311
BC00408=196017,443657,240013
BC00409=195996,443659,293780
BC00410=131872,472570,17
BC00411=131052,467150,17
BC00412=130724,464982,17
BC00413=130724,464982,17
BC00414=130724,464982,17
BC00415=139291,460601,17
BC00416=158742,455857,17
BC00417=161249,454180,17
BC00418=163026,455992,17
BC00419=167469,460520,17
BC00420=167448,460522,17
BC00421=109106,381782,293465
BC00422=110899,386344,284030
BC00423=110899,492791,284030
BC00424=308710,492791,147230
BC00425=398158,484720,4583
BC00426=398158,487298,16212
BC00427=398158,482906,17
BC00428=398158,484456,17
BC00429=398158,481149,17
BC00430=398158,481149,17
BC00431=398158,484456,17
BC00432=398158,484456,17
BC00433=398158,484456,17
BC00434=398158,484456,17
BC00435=398158,491513,1411
BC00436=398158,497594,17653
BC00437=264858,495332,10593
BC00438=251926,517438,69626
BC00439=174889,513712,197000
BC00440=246032,523889,99995
BC00441=249793,518566,85477
BC00442=251297,516426,79670
BC00443=251297,516426,79670
BC00444=251297,516426,79670
BC00445=250422,516425,75433
BC00446=248557,516412,66455
BC00447=247676,516401,62233
BC00448=246171,518541,68040
BC00449=242410,523892,82557
BC00450=199500,464199,40921
BC00451=203261,458848,26404
BC00452=204766,456708,20597
BC00453=204766,456708,20597
BC00454=204766,456708,20597
BC00455=203918,456707,16494
BC00456=202026,456694,7382
BC00457=201172,456683,3293
BC00458=199668,458823,9100
BC00459=195907,464174,23618
BC00460=195886,464176,77385
BC00461=197390,462036,71578
BC00462=197390,518242,269325
BC00463=197390,518242,269325
BC00464=156702,414962,252129
BC00465=132561,353687,302415
BC00466=132561,353687,150779
BC00467=132561,353687,184254
BC00468=132561,353687,188161
BC00469=132561,353687,188161
BC00470=132562,353687,187067
BC00471=132562,353687,187604
BC00472=132562,353688,188102
BC00473=132561,353687,168528
BC00474=132561,353687,132236
BC00475=117787,359154,12124
BC00476=113803,361698,12114
BC00477=106515,366372,12068
BC00478=106515,366372,12068
BC00479=106515,366372,12068
BC00480=106515,366372,12068
BC00481=106515,366372,12068
BC00482=111807,372074,38507
BC00483=155330,418718,512485
BC00484=197390,518242,483003
BC00485=197390,518242,215558
BC00486=259558,439573,183340
BC00487=311189,379628,158993
BC00488=311189,379628,212760
BC00489=311189,379628,212760
BC00490=311189,379628,212760
BC00491=311189,379628,212760
BC00492=311189,379628,212760
BC00493=311189,379628,212760
BC00494=311189,379628,212760
BC00495=311189,379628,212760
BC00496=311189,379628,158993
BC00497=311190,379628,158990
BC00498=311190,379628,158990
BC00499=311190,379628,158990
BC00500=311190,379628,158990
BC00501=311190,379628,158990
BC00502=311190,379628,158990
BC00503=311190,379628,158990
BC00504=311190,379628,158990
BC00505=315633,398424,185896
BC00506=344269,519572,359322
BC00507=148440,436261,427451
BC00508=149297,386225,512925
BC00509=149297,386225,314557
BC00510=149297,386225,267096
BC00511=149297,386225,314557
BC00512=149297,386225,314557
BC00513=149297,386225,314557
BC00514=149297,386225,314557
BC00515=149297,386225,314557
BC00516=149297,386225,314557
BC00517=149297,386225,314557
BC00518=149297,386225,314557
BC00519=199448,515539,1021370
EC00000=-798156,-1296783
EC00001=-798156,-1296783
EC00002=-798156,-1296783
EC00003=-798156,-1296783
EC00004=-798156,-1296783
EC00005=-798156,-1296783
EC00006=-798156,-1296783
EC00007=-798156,-1296783
EC00008=-798156,-1296783
EC00009=-798156,-1296783
EC00010=-798156,-1296783
EC00011=-798156,-1296783
EC00012=-798156,-1296783
EC00013=-798156,-1296783
EC00014=-798156,-1296783
EC00015=-798156,-1296783
EC00016=-798156,-1296783
EC00017=-798156,-1296783
EC00018=-798156,-1296783
EC00019=-798156,-1296783
EC00020=-798156,-1296783
EC00021=-798156,-1296783
EC00022=-798156,-1296783
EC00023=-798156,-1296783
EC00024=-798155,-1296782
EC00025=-798156,-1296783
EC00026=-798156,-1296783
EC00027=-798156,-1296783
EC00028=-798156,-1296783
EC00029=-798156,-1296783
EC00030=-798156,-1296783
EC00031=-798156,-1296783
EC00032=-798156,-1296783
EC00033=-798156,-1296783
EC00034=-798156,-1296783
EC00035=-798156,-1296783
EC00036=-798156,-1296783
EC00037=-798156,-1296783
EC00038=-798156,-1296783
EC00039=-798156,-1296783
EC00040=-798156,-1296783
EC00041=-798156,-1296783
EC00042=-798156,-1296783
EC00043=-798156,-1296783
EC00044=-798156,-1296783
EC00045=-798156,-1296783
EC00046=-798156,-1296783
EC00047=-798156,-1296783
EC00048=-798156,-1296783
EC00049=-798156,-1296783
EC00050=-798156,-1296783
EC00051=-798156,-1296783
EC00052=-798156,-1296783
EC00053=-798156,-1296783
EC00054=-798156,-1296783
EC00055=-798156,-1296783
EC00056=-798156,-1296783
EC00057=-798156,-1296783
EC00058=-798156,-1296783
EC00059=-798156,-1296783
EC00060=-798156,-1296783
EC00061=-798156,-1296783
EC00062=-798156,-1296783
EC00063=-798156,-1296783
EC00064=-798156,-1296783
EC00065=-798156,-1296783
EC00066=-798156,-1296783
EC00067=-798156,-1296783
EC00068=-798156,-1296783
EC00069=-798156,-1296783
EC00070=-798156,-1296783
EC00071=-798156,-1296783
EC00072=-798155,-1296782
EC00073=-798155,-1296782
EC00074=-798155,-1296782
EC00075=-798155,-1296782
EC00076=-798155,-1296782
EC00077=-798155,-1296782
EC00078=-798155,-1296782
EC00079=-798155,-1296782
EC00080=-798155,-1296782
EC00081=-798155,-1296782
EC00082=-798156,-1296783
EC00083=-910680,-1296783
EC00084=-953239,-1296783
EC00085=-960687,-1296783
EC00086=-975524,-1296783
EC00087=-975524,-1296783
EC00088=-975524,-1296783
EC00089=-975524,-1296783
EC00090=-975524,-1296783
EC00091=-975524,-1296783
EC00092=-975524,-1296783
EC00093=-975524,-1296783
EC00094=-975524,-1296783
EC00095=-975524,-1296783
EC00096=-975524,-1296783
EC00097=-975524,-1296783
EC00098=-975524,-1296783
EC00099=-975524,-1296783
EC00100=-975524,-1296783
EC00101=-975524,-1296783
EC00102=-975524,-1296783
EC00103=-975524,-1296783
EC00104=-975524,-1296783
EC00105=-975524,-1296783
EC00106=-975524,-1296783
EC00107=-975524,-1296783
EC00108=-975524,-1296783
EC00109=-975524,-1296783
EC00110=-975524,-1296783
EC00111=-975524,-1296783
EC00112=-975524,-1296783
EC00113=-975521,-1296782
EC00114=-975524,-1296783
EC00115=-975524,-1296783
EC00116=-975524,-1296783
EC00117=-975524,-1296783
EC00118=-975524,-1296783
EC00119=-975524,-1296783
EC00120=-975524,-1296783
EC00121=-975524,-1296783
EC00122=-975524,-1296783
EC00123=-975524,-1296783
EC00124=-975524,-1296783
EC00125=-975524,-1296783
EC00126=-975524,-1296783
EC00127=-975524,-1296783
EC00128=-975524,-1296783
EC00129=-975524,-1296783
EC00130=-975524,-1296783
EC00131=-975524,-1296783
EC00132=-975524,-1296783
EC00133=-975524,-1296783
EC00134=-975524,-1296783
EC00135=-975524,-1296783
EC00136=-975524,-1296783
EC00137=-975524,-1296783
EC00138=-975524,-1296783
EC00139=-975524,-1296783
EC00140=-975524,-1296783
EC00141=-975524,-1296783
EC00142=-975524,-1296783
EC00143=-975521,-1296783
EC00144=-975524,-1296783
EC00145=-975524,-1296783
EC00146=-975521,-1296783
EC00147=-975521,-1296783
EC00148=-975521,-1296783
EC00149=-975521,-1296783
EC00150=-975524,-1296783
EC00151=-975524,-1296783
EC00152=-975524,-1296783
EC00153=-975524,-1296783
EC00154=-975521,-1296781
EC00155=-975524,-1296783
EC00156=-975524,-1296783
EC00157=-975524,-1296783
EC00158=-975524,-1296783
EC00159=-975524,-1296783
EC00160=-975524,-1296783
EC00161=-975524,-1296783
EC00162=-975524,-1296783
EC00163=-975524,-1296783
EC00164=-975524,-1296783
EC00165=-975524,-1296783
EC00166=-975524,-1296783
EC00167=-975524,-1296783
EC00168=-975524,-1296783
EC00169=-975524,-1296783
EC00170=-975524,-1296783
EC00171=-975524,-1296783
EC00172=-975524,-1296783
EC00173=-975524,-1296783
EC00174=-975524,-1296783
EC00175=-975524,-1296783
EC00176=-975524,-1296783
EC00177=-975524,-1296783
EC00178=-975524,-1296783
EC00179=-975524,-1296783
EC00180=-975524,-1296783
EC00181=-975524,-1296783
EC00182=-975524,-1296783
EC00183=-975524,-1296783
EC00184=-975524,-1296783
EC00185=-975524,-1296783
EC00186=-975524,-1296783
EC00187=-975524,-1296783
EC00188=-975524,-1296783
EC00189=-975524,-1296783
EC00190=-975524,-1296783
EC00191=-975524,-1296783
EC00192=-975524,-1296783
EC00193=-975524,-1296783
EC00194=-975524,-1296783
EC00195=-975524,-1296783
EC00196=-975524,-1296783
EC00197=-975524,-1296783
EC00198=-975524,-1296783
EC00199=-975524,-1296783
EC00200=-975524,-1296783
EC00201=-975524,-1296783
EC00202=-975524,-1296783
EC00203=-975524,-1296783
EC00204=-975524,-1296783
EC00205=-975524,-1296783
EC00206=-975524,-1296783
EC00207=-975524,-1296783
EC00208=-975524,-1296783
EC00209=-975524,-1296783
EC00210=-975512,-1296779
EC00211=-975524,-1296783
EC00212=-975524,-1296783
EC00213=-975515,-1296780
EC00214=-975524,-1296783
EC00215=-975524,-1296783
EC00216=-975521,-1296782
EC00217=-975524,-1296783
EC00218=-975524,-1296783
EC00219=-975524,-1296783
EC00220=-975524,-1296783
EC00221=-975524,-1296783
EC00222=-975524,-1296783
EC00223=-975524,-1296783
EC00224=-975524,-1296783
EC00225=-975524,-1296783
EC00226=-975524,-1296783
EC00227=-975524,-1296783
EC00228=-975524,-1296783
EC00229=-975524,-1296783
EC00230=-975524,-1296783
EC00231=-975524,-1296783
EC00232=-975524,-1296783
EC00233=-975524,-1296783
EC00234=-975524,-1296783
EC00235=-975524,-1296783
EC00236=-975524,-1296783
EC00237=-975524,-1296783
EC00238=-798156,-1296783
EC00239=-798156,-1296783
EC00240=-798156,-1296783
EC00241=-798156,-1296783
EC00242=-798156,-1296783
EC00243=-798156,-1296783
EC00244=-798156,-1296783
EC00245=-798156,-1296783
EC00246=-798156,-1296783
EC00247=-798156,-1296783
EC00248=-798156,-1296783
EC00249=-798156,-1296783
EC00250=-798156,-1296783
EC00251=-798156,-1296783
EC00252=-798156,-1296783
EC00253=-798156,-1296783
EC00254=-798156,-1296783
EC00255=-798156,-1296783
EC00256=-798156,-1296783
EC00257=-798156,-1296783
EC00258=-798156,-1296783
EC00259=-798156,-1296783
EC00260=-798156,-1296783
EC00261=-798156,-1296783
EC00262=-798156,-1296783
EC00263=-798156,-1296783
EC00264=-798156,-1296783
EC00265=-798156,-1296783
EC00266=-798156,-1296783
EC00267=-798156,-1296783
EC00268=-798156,-1296783
EC00269=-798156,-1296783
EC00270=-798153,-1296780
EC00271=-798155,-1296782
EC00272=-798155,-1296782
EC00273=-798155,-1296782
EC00274=-798155,-1296782
EC00275=-798156,-1296783
EC00276=-798156,-1296783
EC00277=-798156,-1296783
EC00278=-798156,-1296783
EC00279=-798156,-1296783
EC00280=-798156,-1296783
EC00281=-798156,-1296783
EC00282=-798156,-1296783
EC00283=-798156,-1296783
EC00284=-798156,-1296783
EC00285=-798156,-1296783
EC00286=-798156,-1296783
EC00287=-798156,-1296783
EC00288=-798156,-1296783
EC00289=-798156,-1296783
EC00290=-798156,-1296783
EC00291=-798156,-1296783
EC00292=-798156,-1296783
EC00293=-798156,-1296783
EC00294=-798156,-1296783
EC00295=-798156,-1296783
EC00296=-798156,-1296783
EC00297=-798156,-1296783
EC00298=-798156,-1296783
EC00299=-798156,-1296783
EC00300=-798156,-1296783
EC00301=-798156,-1296783
EC00302=-798156,-1296783
EC00303=-798156,-1296783
EC00304=-798156,-1296783
EC00305=-798156,-1296783
EC00306=-798156,-1296783
EC00307=-798156,-1296783
EC00308=-798156,-1296783
EC00309=-798156,-1296783
EC00310=-798156,-1296783
EC00311=-798156,-1296783
EC00312=-798156,-1296783
EC00313=-798156,-1296783
EC00314=-798156,-1296783
EC00315=-798156,-1296783
EC00316=-798156,-1296783
EC00317=-798156,-1296783
EC00318=-798156,-1296783
EC00319=-798156,-1296783
EC00320=-798156,-1296783
EC00321=-798156,-1296783
EC00322=-798156,-1296783
EC00323=-798156,-1296783
EC00324=-798156,-1296783
EC00325=-798156,-1296783
EC00326=-798156,-1296783
EC00327=-798156,-1296783
EC00328=-798156,-1296783
EC00329=-798156,-1296783
EC00330=-798156,-1296783
EC00331=-798156,-1296783
EC00332=-798156,-1296783
EC00333=-798156,-1296783
EC00334=-798156,-1296783
EC00335=-798156,-1296783
EC00336=-798156,-1296783
EC00337=-798156,-1296783
EC00338=-798156,-1296783
EC00339=-798156,-1296783
EC00340=-798156,-1296783
EC00341=-798156,-1296783
EC00342=-798156,-1296783
EC00343=-798156,-1296783
EC00344=-798156,-1296783
EC00345=-798156,-1296783
EC00346=-798156,-1296783
EC00347=-798156,-1296783
EC00348=-798156,-1296783
EC00349=-798156,-1296783
EC00350=-798156,-1296783
EC00351=-798156,-1296783
EC00352=-798156,-1296783
EC00353=-798156,-1296783
EC00354=-798156,-1296783
EC00355=-798156,-1296783
EC00356=-798156,-1296783
EC00357=-798156,-1296783
EC00358=-798156,-1296783
EC00359=-798156,-1296783
EC00360=-798156,-1296783
EC00361=-798156,-1296783
EC00362=-798156,-1296783
EC00363=-798156,-1296783
EC00364=-798156,-1296783
EC00365=-798156,-1296783
EC00366=-798156,-1296783
EC00367=-798156,-1296783
EC00368=-798156,-1296783
EC00369=-798156,-1296783
EC00370=-798156,-1296783
EC00371=-798156,-1296783
EC00372=-798156,-1296783
EC00373=-798156,-1296783
EC00374=-798156,-1296783
EC00375=-798156,-1296783
EC00376=-798156,-1296783
EC00377=-798156,-1296783
EC00378=-798156,-1296783
EC00379=-798156,-1296783
EC00380=-798156,-1296783
EC00381=-798156,-1296783
EC00382=-798156,-1296783
EC00383=-798156,-1296783
EC00384=-798156,-1296783
EC00385=-798156,-1296783
EC00386=-798156,-1296783
EC00387=-798156,-1296783
EC00388=-798156,-1296783
EC00389=-798156,-1296783
EC00390=-798156,-1296783
EC00391=-798156,-1296783
EC00392=-798156,-1296783
EC00393=-798156,-1296783
EC00394=-798156,-1296783
EC00395=-798156,-1296783
EC00396=-798156,-1296783
EC00397=-798156,-1296783
EC00398=-798156,-1296783
EC00399=-798156,-1296783
EC00400=-798156,-1296783
EC00401=-798156,-1296783
EC00402=-798156,-1296783
EC00403=-798156,-1296783
EC00404=-798156,-1296783
EC00405=-798156,-1296783
EC00406=-798156,-1296783
EC00407=-798156,-1296783
EC00408=-798156,-1296783
EC00409=-798156,-1296783
EC00410=-798156,-1296783
EC00411=-798156,-1296783
EC00412=-798156,-1296783
EC00413=-798156,-1296783
EC00414=-798156,-1296783
EC00415=-798156,-1296783
EC00416=-798156,-1296783
EC00417=-798156,-1296783
EC00418=-798156,-1296783
EC00419=-798156,-1296783
EC00420=-798156,-1296783
EC00421=-798156,-1296783
EC00422=-798156,-1296783
EC00423=-798156,-1296783
EC00424=-798156,-1296783
EC00425=-798156,-1296783
EC00426=-798156,-1296783
EC00427=-798156,-1296783
EC00428=-798156,-1296783
EC00429=-798156,-1296783
EC00430=-798156,-1296783
EC00431=-798156,-1296783
EC00432=-798156,-1296783
EC00433=-798156,-1296783
EC00434=-798156,-1296783
EC00435=-798156,-1296783
EC00436=-798156,-1296783
EC00437=-798156,-1296783
EC00438=-798156,-1296783
EC00439=-798156,-1296783
EC00440=-798156,-1296783
EC00441=-798156,-1296783
EC00442=-798156,-1296783
EC00443=-798156,-1296783
EC00444=-798156,-1296783
EC00445=-798156,-1296783
EC00446=-798156,-1296783
EC00447=-798156,-1296783
EC00448=-798156,-1296783
EC00449=-798156,-1296783
EC00450=-798156,-1296783
EC00451=-798156,-1296783
EC00452=-798156,-1296783
EC00453=-798156,-1296783
EC00454=-798156,-1296783
EC00455=-798156,-1296783
EC00456=-798156,-1296783
EC00457=-798156,-1296783
EC00458=-798156,-1296783
EC00459=-798156,-1296783
EC00460=-798156,-1296783
EC00461=-798156,-1296783
EC00462=-798156,-1296783
EC00463=-798156,-1296783
EC00464=-798155,-1296783
EC00465=-798156,-1296783
EC00466=-798156,-1296783
EC00467=-798156,-1296783
EC00468=-798156,-1296783
EC00469=-798156,-1296783
EC00470=-798154,-1296782
EC00471=-798155,-1296782
EC00472=-798155,-1296782
EC00473=-798156,-1296783
EC00474=-798156,-1296783
EC00475=-798156,-1296783
EC00476=-798156,-1296783
EC00477=-798156,-1296783
EC00478=-798156,-1296783
EC00479=-798156,-1296783
EC00480=-798156,-1296783
EC00481=-798156,-1296783
EC00482=-798156,-1296783
EC00483=-798156,-1296783
EC00484=-798156,-1296783
EC00485=-798156,-1296783
EC00486=-798156,-1296783
EC00487=-798156,-1296783
EC00488=-798156,-1296783
EC00489=-798156,-1296783
EC00490=-798156,-1296783
EC00491=-798156,-1296783
EC00492=-798156,-1296783
EC00493=-798156,-1296783
EC00494=-798156,-1296783
EC00495=-798156,-1296783
EC00496=-798156,-1296783
EC00497=-798155,-1296782
EC00498=-798155,-1296782
EC00499=-798155,-1296782
EC00500=-798155,-1296782
EC00501=-798155,-1296782
EC00502=-798155,-1296782
EC00503=-798155,-1296782
EC00504=-798155,-1296782
EC00505=-798155,-1296782
EC00506=-798156,-1296783
EC00507=-798156,-1296783
EC00508=-798156,-1296783
EC00509=-798156,-1296783
EC00510=-798156,-1296783
EC00511=-798156,-1296783
EC00512=-798156,-1296783
EC00513=-798156,-1296783
EC00514=-798156,-1296783
EC00515=-798156,-1296783
EC00516=-798156,-1296783
EC00517=-798156,-1296783
EC00518=-798156,-1296783
EC00519=-798155,-1296782
///POSTYPE BASE
///RECTAN
///RCONF 0,0,0,0,1,0,0,0,0,0,0,0,0,0,0,0,0,0,0,0,0,0,0,0
P00006=2.006,1.622,-0.565,0.0000,0.0000,0.0000
P00021=0.073,2.058,-0.109,0.0000,0.0000,0.0000
P00022=2.006,1.622,-0.565,0.0000,0.0000,0.0000
///RCONF 0,0,0,0,0,0,0,0,0,0,0,0,0,0,0,0,0,0,0,0,0,0,0,0
P00023=-2.957,-4.083,2.762,0.0000,0.0000,0.0000
P00024=-1.466,-0.226,-0.419,0.0000,0.0000,0.0000
P00025=3.643,0.007,-2.585,0.0000,0.0000,0.0000
P00026=2.644,0.055,-2.583,0.0000,0.0000,0.0000
P00027=2.278,0.099,-4.210,0.0000,0.0000,0.0000
P00031=-0.170,0.039,-0.647,0.0000,0.0000,0.0000
P00032=-0.423,0.157,3.222,0.0000,0.0000,0.0000
P00041=-0.109,0.014,0.966,0.0000,0.0000,0.0000
P00042=-0.220,0.371,-0.613,0.0000,0.0000,0.0000
P00043=-0.179,-5.890,-3.227,0.0000,0.0000,0.0000
P00044=-8.560,-7.557,-5.232,0.0000,0.0000,0.0000
P00045=-8.836,-6.632,-1.438,0.0000,0.0000,0.0000
P00046=-7.725,-0.107,-2.878,0.0000,0.0000,0.0000
P00088=-8.588,-0.108,-11.097,0.0000,0.0000,0.0000
P00089=5.931,-12.286,-8.772,0.0000,0.0000,0.0000
P00090=-14.057,13.261,-6.464,0.0000,0.0000,0.0000
//INST
///DATE 2024/11/19 20:21
///ATTR SC,RW
///GROUP1 RB1,BS1
///GROUP2 ST1
NOP
'OK_r2_O57-69(2)(90,0)2
'Down
SFTOF3D
MOVJ C00000 BC00000 VJ=100.00  +MOVJ EC00000 VJ=100.00
MOVL C00001 BC00001 V=400.0  +MOVJ EC00001 VJ=100.00
SMOVL C00002 BC00002 V=166.7  +MOVJ EC00002
SREFP 3 C00003 BC00003  +REFP EC00003
CALL JOB:SEARCH-R1-S13D
SET P026 P006
SFTON3D P026
SMOVL C00004 BC00004 V=166.7  +MOVJ EC00004
SREFP 3 C00005 BC00005  +REFP EC00005
CALL JOB:SEARCH-R1-S13D
SET P026 P006
SFTON3D P026
SMOVL C00006 BC00006 V=166.7  +MOVJ EC00006
MOVL C00007 BC00007 V=400.0  +MOVJ EC00007 VJ=100.00
MOVL C00008 BC00008 V=1000.0  +MOVJ EC00008 VJ=100.00
'Path S3529
SFTOF3D
MOVJ C00009 BC00009 VJ=100.00  +MOVJ EC00009 VJ=100.00
MOVL C00010 BC00010 V=400.0  +MOVJ EC00010 VJ=100.00
SMOVL C00011 BC00011 V=166.7  +MOVJ EC00011
SREFP 3 C00012 BC00012  +REFP EC00012
CALL JOB:SEARCH-R1-S13D
SET P027 P006
SFTON3D P027
SMOVL C00013 BC00013 V=166.7  +MOVJ EC00013
SREFP 3 C00014 BC00014  +REFP EC00014
CALL JOB:SEARCH-R1-S13D
SET P027 P006
SFTON3D P027
SMOVL C00015 BC00015 V=166.7  +MOVJ EC00015
MOVL C00016 BC00016 V=400.0  +MOVJ EC00016 VJ=100.00
MOVL C00017 BC00017 V=1000.0  +MOVJ EC00017 VJ=100.00
MOVL C00018 BC00018 V=1000.0  +MOVJ EC00018 VJ=100.00
'Path S3530
SFTOF3D
MOVJ C00019 BC00019 VJ=100.00  +MOVJ EC00019 VJ=100.00
MOVL C00020 BC00020 V=400.0  +MOVJ EC00020 VJ=100.00
SMOVL C00021 BC00021 V=166.7  +MOVJ EC00021
SREFP 3 C00022 BC00022  +REFP EC00022
CALL JOB:SEARCH-R1-S13D
SET P022 P006
SFTON3D P022
SMOVL C00023 BC00023 V=166.7  +MOVJ EC00023
SREFP 3 C00024 BC00024  +REFP EC00024
CALL JOB:SEARCH-R1-S13D
SET P022 P006
SFTON3D P022
SMOVL C00025 BC00025 V=166.7  +MOVJ EC00025
SFTOF3D
MOVL C00026 BC00026 V=1000.0  +MOVJ EC00026 VJ=100.00
SMOVL C00027 BC00027 V=1000.0  +MOVJ EC00027
SMOVL C00028 BC00028 V=166.7  +MOVJ EC00028
SREFP 3 C00029 BC00029  +REFP EC00029
CALL JOB:SEARCH-R1-S13D
SET P088 P006
SFTON3D P088
SMOVL C00030 BC00030 V=166.7  +MOVJ EC00030
SMOVL C00031 BC00031 V=166.7  +MOVJ EC00031
SMOVL C00032 BC00032 V=166.7  +MOVJ EC00032
SREFP 3 C00033 BC00033  +REFP EC00033
CALL JOB:SEARCH-R1-S13D
SET P088 P006
SFTON3D P088
SMOVL C00034 BC00034 V=166.7  +MOVJ EC00034
SFTOF3D
SMOVL C00035 BC00035 V=1000.0  +MOVJ EC00035
MOVJ C00036 BC00036 VJ=100.00  +MOVJ EC00036 VJ=100.00
MOVJ C00037 BC00037 VJ=100.00  +MOVJ EC00037 VJ=100.00
MOVL C00038 BC00038 V=400.0  +MOVJ EC00038 VJ=100.00
SMOVL C00039 BC00039 V=133.3  +MOVJ EC00039
SREFP 3 C00040 BC00040  +REFP EC00040
CALL JOB:SEARCH-R1-S13D
SET P021 P006
SFTON3D P021
SMOVL C00041 BC00041 V=166.7  +MOVJ EC00041
SREFP 3 C00042 BC00042  +REFP EC00042
CALL JOB:SEARCH-R1-S13D
SET P021 P006
SFTON3D P021
SMOVL C00043 BC00043 V=166.7  +MOVJ EC00043
SMOVL C00044 BC00044 V=166.7  +MOVJ EC00044
SREFP 3 C00045 BC00045  +REFP EC00045
CALL JOB:SEARCH-R1-S13D
SET P021 P006
SFTON3D P021
SMOVL C00046 BC00046 V=166.7  +MOVJ EC00046
MOVL C00047 BC00047 V=400.0  +MOVJ EC00047 VJ=100.00
MOVL C00048 BC00048 V=1000.0  +MOVJ EC00048 VJ=100.00
MOVJ C00049 BC00049 VJ=100.00  +MOVJ EC00049 VJ=100.00
MOVJ C00050 BC00050 VJ=100.00  +MOVJ EC00050 VJ=100.00
'Path S3538
SFTOF3D
MOVJ C00051 BC00051 VJ=100.00  +MOVJ EC00051 VJ=100.00
MOVL C00052 BC00052 V=400.0  +MOVJ EC00052 VJ=100.00
SMOVL C00053 BC00053 V=166.7  +MOVJ EC00053
SREFP 3 C00054 BC00054  +REFP EC00054
CALL JOB:SEARCH-R1-S13D
SET P032 P006
SFTON3D P032
SMOVL C00055 BC00055 V=166.7  +MOVJ EC00055
SREFP 3 C00056 BC00056  +REFP EC00056
CALL JOB:SEARCH-R1-S13D
SET P032 P006
SFTON3D P032
SMOVL C00057 BC00057 V=166.7  +MOVJ EC00057
SFTOF3D
MOVL C00058 BC00058 V=400.0  +MOVJ EC00058 VJ=100.00
MOVL C00059 BC00059 V=1000.0  +MOVJ EC00059 VJ=100.00
MOVJ C00060 BC00060 VJ=100.00  +MOVJ EC00060 VJ=100.00
MOVJ C00061 BC00061 VJ=100.00  +MOVJ EC00061 VJ=100.00
COMM PAUSE
COMM MOVJ C00062 BC00062 VJ=100.00  +MOVJ EC00062 VJ=100.00
COMM SMOVL C00063 BC00063 V=1000.0  +MOVJ EC00063
COMM SMOVL C00064 BC00064 V=166.7  +MOVJ EC00064
COMM SREFP 3 C00065 BC00065  +REFP EC00065
COMM CALL JOB:SEARCH-R1-S13D
COMM SET P089 P006
COMM SFTON3D P089
COMM SMOVL C00066 BC00066 V=166.7  +MOVJ EC00066
COMM SMOVL C00067 BC00067 V=166.7  +MOVJ EC00067
COMM SMOVL C00068 BC00068 V=166.7  +MOVJ EC00068
COMM SREFP 3 C00069 BC00069  +REFP EC00069
COMM CALL JOB:SEARCH-R1-S13D
COMM SET P089 P006
COMM SFTON3D P089
COMM SMOVL C00070 BC00070 V=166.7  +MOVJ EC00070
COMM SFTOF3D
SMOVL C00071 BC00071 V=1000.0  +MOVJ EC00071
SMOVL C00072 BC00072 V=1000.0  +MOVJ EC00072
SMOVL C00073 BC00073 V=166.7  +MOVJ EC00073
SREFP 3 C00074 BC00074  +REFP EC00074
CALL JOB:SEARCH-R1-S13D
SET P090 P006
SFTON3D P090
SMOVL C00075 BC00075 V=166.7  +MOVJ EC00075
SREFP 3 C00076 BC00076  +REFP EC00076
CALL JOB:SEARCH-R1-S13D
SET P090 P006
SFTON3D P090
SMOVL C00077 BC00077 V=166.7  +MOVJ EC00077
SMOVL C00078 BC00078 V=166.7  +MOVJ EC00078
SREFP 3 C00079 BC00079  +REFP EC00079
CALL JOB:SEARCH-R1-S13D
SET P090 P006
SFTON3D P090
SMOVL C00080 BC00080 V=250.0  +MOVJ EC00080
SFTOF3D
SMOVL C00081 BC00081 V=1000.0  +MOVJ EC00081
SMOVL C00082 BC00082 V=1000.0  +MOVJ EC00082
MOVJ C00083 BC00083 VJ=100.00  +MOVJ EC00083 VJ=100.00
'Up
MOVJ C00084 BC00084 VJ=100.00  +MOVJ EC00084 VJ=100.00
MOVJ C00085 BC00085 VJ=100.00  +MOVJ EC00085 VJ=100.00
'Path S3539
SFTOF3D
MOVJ C00086 BC00086 VJ=100.00  +MOVJ EC00086 VJ=100.00
MOVL C00087 BC00087 V=400.0  +MOVJ EC00087 VJ=100.00
SMOVL C00088 BC00088 V=100.0  +MOVJ EC00088
SREFP 3 C00089 BC00089  +REFP EC00089
CALL JOB:SEARCH-R1-S13D
SET P046 P006
SFTON3D P046
SMOVL C00090 BC00090 V=100.0  +MOVJ EC00090
SREFP 3 C00091 BC00091  +REFP EC00091
CALL JOB:SEARCH-R1-S13D
SET P046 P006
SFTON3D P046
SMOVL C00092 BC00092 V=100.0  +MOVJ EC00092
MOVL C00093 BC00093 V=400.0  +MOVJ EC00093 VJ=100.00
MOVL C00094 BC00094 V=1000.0  +MOVJ EC00094 VJ=100.00
'Path S3540
SFTOF3D
MOVJ C00095 BC00095 VJ=100.00  +MOVJ EC00095 VJ=100.00
MOVL C00096 BC00096 V=400.0  +MOVJ EC00096 VJ=100.00
SMOVL C00097 BC00097 V=100.0  +MOVJ EC00097
SREFP 3 C00098 BC00098  +REFP EC00098
CALL JOB:SEARCH-R1-S13D
SET P045 P006
SFTON3D P045
SMOVL C00099 BC00099 V=100.0  +MOVJ EC00099
SREFP 3 C00100 BC00100  +REFP EC00100
CALL JOB:SEARCH-R1-S13D
SET P045 P006
SFTON3D P045
SMOVL C00101 BC00101 V=100.0  +MOVJ EC00101
SREFP 3 C00102 BC00102  +REFP EC00102
CALL JOB:SEARCH-R1-S13D
SET P045 P006
SFTON3D P045
SMOVL C00103 BC00103 V=100.0  +MOVJ EC00103
MOVL C00104 BC00104 V=400.0  +MOVJ EC00104 VJ=100.00
MOVL C00105 BC00105 V=1000.0  +MOVJ EC00105 VJ=100.00
MOVL C00106 BC00106 V=1000.0  +MOVJ EC00106 VJ=100.00
MOVJ C00107 BC00107 VJ=100.00  +MOVJ EC00107 VJ=50.00
SFTOF3D
MOVJ C00108 BC00108 VJ=100.00  +MOVJ EC00108 VJ=50.00
MOVJ C00109 BC00109 VJ=100.00  +MOVJ EC00109 VJ=100.00
MOVL C00110 BC00110 V=400.0  +MOVJ EC00110 VJ=100.00
SMOVL C00111 BC00111 V=100.0  +MOVJ EC00111
SREFP 3 C00112 BC00112  +REFP EC00112
CALL JOB:SEARCH-R1-S13D
SET P043 P006
SFTON3D P043
SMOVL C00113 BC00113 V=100.0  +MOVJ EC00113
SREFP 3 C00114 BC00114  +REFP EC00114
CALL JOB:SEARCH-R1-S13D
SET P043 P006
SFTON3D P043
SMOVL C00115 BC00115 V=100.0  +MOVJ EC00115
SREFP 3 C00116 BC00116  +REFP EC00116
CALL JOB:SEARCH-R1-S13D
SET P043 P006
SFTON3D P043
SMOVL C00117 BC00117 V=100.0  +MOVJ EC00117
MOVL C00118 BC00118 V=400.0  +MOVJ EC00118 VJ=100.00
MOVL C00119 BC00119 V=1000.0  +MOVJ EC00119 VJ=100.00
'Path S3543
SFTOF3D
MOVJ C00120 BC00120 VJ=100.00  +MOVJ EC00120 VJ=100.00
MOVL C00121 BC00121 V=400.0  +MOVJ EC00121 VJ=100.00
SMOVL C00122 BC00122 V=100.0  +MOVJ EC00122
SREFP 3 C00123 BC00123  +REFP EC00123
CALL JOB:SEARCH-R1-S13D
SET P042 P006
SFTON3D P042
SMOVL C00124 BC00124 V=100.0  +MOVJ EC00124
SREFP 3 C00125 BC00125  +REFP EC00125
CALL JOB:SEARCH-R1-S13D
SET P042 P006
SFTON3D P042
SMOVL C00126 BC00126 V=100.0  +MOVJ EC00126
SREFP 3 C00127 BC00127  +REFP EC00127
CALL JOB:SEARCH-R1-S13D
SET P042 P006
SFTON3D P042
SMOVL C00128 BC00128 V=100.0  +MOVJ EC00128
MOVL C00129 BC00129 V=1000.0  +MOVJ EC00129 VJ=100.00
'Path S3544
SFTOF3D
MOVJ C00130 BC00130 VJ=100.00  +MOVJ EC00130 VJ=100.00
MOVL C00131 BC00131 V=400.0  +MOVJ EC00131 VJ=100.00
SMOVL C00132 BC00132 V=100.0  +MOVJ EC00132
SREFP 3 C00133 BC00133  +REFP EC00133
CALL JOB:SEARCH-R1-S13D
SET P041 P006
SFTON3D P041
SMOVL C00134 BC00134 V=100.0  +MOVJ EC00134
SREFP 3 C00135 BC00135  +REFP EC00135
CALL JOB:SEARCH-R1-S13D
SET P041 P006
SFTON3D P041
SMOVL C00136 BC00136 V=100.0  +MOVJ EC00136
SREFP 3 C00137 BC00137  +REFP EC00137
CALL JOB:SEARCH-R1-S13D
SET P041 P006
SFTON3D P041
SMOVL C00138 BC00138 V=100.0  +MOVJ EC00138
MOVL C00139 BC00139 V=400.0  +MOVJ EC00139 VJ=100.00
MOVL C00140 BC00140 V=1000.0  +MOVJ EC00140 VJ=100.00
'Path W3545
SFTOF3D
SFTON3D P041
MOVJ C00141 BC00141 VJ=100.00  +MOVJ EC00141 VJ=100.00
SMOVL C00142 BC00142 V=400.0  +MOVJ EC00142
SMOVL C00143 BC00143 V=133.3 PL=0  +MOVJ EC00143
SREFP 1 C00144 BC00144  +REFP EC00144
SREFP 2 C00145 BC00145  +REFP EC00145
MACRO1 MJ#(0) ARGF9
ARCON
SWVON WEV#(61)
SMOVL C00146 BC00146 V=6.7  +MOVJ EC00146
SMOVL C00147 BC00147 V=6.7  +MOVJ EC00147
SMOVL C00148 BC00148 V=6.7  +MOVJ EC00148
ARCOF
SWVOF
SMOVL C00149 BC00149 V=400.0  +MOVJ EC00149
SMOVL C00150 BC00150 V=1000.0  +MOVJ EC00150
SFTOF3D
'Path W3546
SFTOF3D
SFTON3D P042
MOVJ C00151 BC00151 VJ=100.00  +MOVJ EC00151 VJ=100.00
MOVJ C00152 BC00152 VJ=100.00  +MOVJ EC00152 VJ=100.00
SMOVL C00153 BC00153 V=400.0  +MOVJ EC00153
SMOVL C00154 BC00154 V=133.3 PL=0  +MOVJ EC00154
SREFP 1 C00155 BC00155  +REFP EC00155
SREFP 2 C00156 BC00156  +REFP EC00156
MACRO1 MJ#(0) ARGF14
ARCON
SMOVL C00157 BC00157 V=8.3  +MOVJ EC00157
SMOVL C00158 BC00158 V=8.3  +MOVJ EC00158
SMOVL C00159 BC00159 V=8.3  +MOVJ EC00159
ARCOF
SMOVL C00160 BC00160 V=400.0  +MOVJ EC00160
SMOVL C00161 BC00161 V=333.3  +MOVJ EC00161
SFTOF3D
MOVJ C00162 BC00162 VJ=100.00  +MOVJ EC00162 VJ=100.00
'Path W3547
SFTOF3D
SFTON3D P043
MOVJ C00163 BC00163 VJ=100.00  +MOVJ EC00163 VJ=100.00
MOVJ C00164 BC00164 VJ=100.00  +MOVJ EC00164 VJ=100.00
SMOVL C00165 BC00165 V=400.0  +MOVJ EC00165
SMOVL C00166 BC00166 V=133.3 PL=0  +MOVJ EC00166
SREFP 1 C00167 BC00167  +REFP EC00167
SREFP 2 C00168 BC00168  +REFP EC00168
MACRO1 MJ#(0) ARGF14
ARCON
SMOVL C00169 BC00169 V=8.3  +MOVJ EC00169
SMOVL C00170 BC00170 V=8.3  +MOVJ EC00170
ARCOF
SMOVL C00171 BC00171 V=400.0  +MOVJ EC00171
SMOVL C00172 BC00172 V=1000.0  +MOVJ EC00172
SMOVL C00173 BC00173 V=1000.0  +MOVJ EC00173
SFTOF3D
'NIE SPAWAMY
COMM 'Path W3548
COMM SFTOF3D
COMM SFTON3D P044
COMM MOVJ C00174 BC00174 VJ=100.00  +MOVJ EC00174 VJ=100.00
COMM SMOVL C00175 BC00175 V=400.0  +MOVJ EC00175
COMM SMOVL C00176 BC00176 V=100.0 PL=0  +MOVJ EC00176
COMM SREFP 1 C00177 BC00177  +REFP EC00177
COMM SREFP 2 C00178 BC00178  +REFP EC00178
COMM MACRO1 MJ#(0) ARGF0
COMM ARCON
COMM SMOVL C00179 BC00179 V=10.0  +MOVJ EC00179
COMM SMOVL C00180 BC00180 V=10.0  +MOVJ EC00180
COMM SMOVL C00181 BC00181 V=10.0  +MOVJ EC00181
COMM SMOVL C00182 BC00182 V=10.0  +MOVJ EC00182
COMM SMOVL C00183 BC00183 V=10.0  +MOVJ EC00183
COMM SMOVL C00184 BC00184 V=10.0  +MOVJ EC00184
COMM SMOVL C00185 BC00185 V=10.0  +MOVJ EC00185
COMM SMOVL C00186 BC00186 V=10.0  +MOVJ EC00186
COMM SMOVL C00187 BC00187 V=10.0  +MOVJ EC00187
COMM SMOVL C00188 BC00188 V=10.0  +MOVJ EC00188
COMM SMOVL C00189 BC00189 V=10.0  +MOVJ EC00189
COMM SMOVL C00190 BC00190 V=10.0  +MOVJ EC00190
COMM SMOVL C00191 BC00191 V=10.0  +MOVJ EC00191
COMM SMOVL C00192 BC00192 V=10.0  +MOVJ EC00192
COMM SMOVL C00193 BC00193 V=10.0  +MOVJ EC00193
COMM SMOVL C00194 BC00194 V=10.0  +MOVJ EC00194
COMM SMOVL C00195 BC00195 V=10.0  +MOVJ EC00195
COMM SMOVL C00196 BC00196 V=10.0  +MOVJ EC00196
COMM SMOVL C00197 BC00197 V=10.0  +MOVJ EC00197
COMM SMOVL C00198 BC00198 V=10.0  +MOVJ EC00198
COMM SMOVL C00199 BC00199 V=10.0  +MOVJ EC00199
COMM SMOVL C00200 BC00200 V=10.0  +MOVJ EC00200
COMM SMOVL C00201 BC00201 V=10.0  +MOVJ EC00201
COMM SMOVL C00202 BC00202 V=10.0  +MOVJ EC00202
COMM SMOVL C00203 BC00203 V=10.0  +MOVJ EC00203
COMM ARCOF
COMM SMOVL C00204 BC00204 V=400.0  +MOVJ EC00204
COMM SMOVL C00205 BC00205 V=1000.0  +MOVJ EC00205
COMM SFTOF3D
'Path W3549
SFTOF3D
MOVJ C00206 BC00206 VJ=100.00  +MOVJ EC00206 VJ=100.00
MOVJ C00207 BC00207 VJ=100.00  +MOVJ EC00207 VJ=100.00
SFTON3D P045
MOVJ C00208 BC00208 VJ=100.00  +MOVJ EC00208 VJ=100.00
SMOVL C00209 BC00209 V=400.0  +MOVJ EC00209
SMOVL C00210 BC00210 V=100.0 PL=0  +MOVJ EC00210
SREFP 1 C00211 BC00211  +REFP EC00211
SREFP 2 C00212 BC00212  +REFP EC00212
MACRO1 MJ#(0) ARGF14
ARCON
SMOVL C00213 BC00213 V=8.3  +MOVJ EC00213
SMOVL C00214 BC00214 V=8.3  +MOVJ EC00214
SMOVL C00215 BC00215 V=8.3  +MOVJ EC00215
SMOVL C00216 BC00216 V=8.3  +MOVJ EC00216
SMOVL C00217 BC00217 V=8.3  +MOVJ EC00217
ARCOF
SMOVL C00218 BC00218 V=400.0  +MOVJ EC00218
SMOVL C00219 BC00219 V=1000.0  +MOVJ EC00219
SMOVL C00220 BC00220 V=1000.0  +MOVJ EC00220
MOVJ C00221 BC00221 VJ=100.00  +MOVJ EC00221 VJ=50.00
SFTOF3D
'Path W3550
SFTOF3D
SFTON3D P046
MOVJ C00222 BC00222 VJ=100.00  +MOVJ EC00222 VJ=100.00
MOVJ C00223 BC00223 VJ=100.00  +MOVJ EC00223 VJ=100.00
SMOVL C00224 BC00224 V=400.0  +MOVJ EC00224
SMOVL C00225 BC00225 V=100.0 PL=0  +MOVJ EC00225
SREFP 1 C00226 BC00226  +REFP EC00226
SREFP 2 C00227 BC00227  +REFP EC00227
MACRO1 MJ#(0) ARGF14
ARCON
SMOVL C00228 BC00228 V=8.3  +MOVJ EC00228
SMOVL C00229 BC00229 V=8.3  +MOVJ EC00229
SMOVL C00230 BC00230 V=8.3  +MOVJ EC00230
SMOVL C00231 BC00231 V=8.3  +MOVJ EC00231
SMOVL C00232 BC00232 V=8.3  +MOVJ EC00232
SMOVL C00233 BC00233 V=8.3  +MOVJ EC00233
ARCOF
SMOVL C00234 BC00234 V=400.0  +MOVJ EC00234
SMOVL C00235 BC00235 V=1000.0  +MOVJ EC00235
SFTOF3D
MOVJ C00236 BC00236 VJ=100.00  +MOVJ EC00236 VJ=100.00
MOVJ C00237 BC00237 VJ=100.00  +MOVJ EC00237 VJ=100.00
MOVJ C00238 BC00238 VJ=100.00  +MOVJ EC00238 VJ=100.00
'Down
'Path W3551
SFTOF3D
MOVJ C00239 BC00239 VJ=100.00  +MOVJ EC00239 VJ=100.00
MOVL C00240 BC00240 V=400.0  +MOVJ EC00240 VJ=100.00
SFTON3D P032
SMOVL C00241 BC00241 V=100.0 PL=0  +MOVJ EC00241
SREFP 1 C00242 BC00242  +REFP EC00242
SREFP 2 C00243 BC00243  +REFP EC00243
MACRO1 MJ#(0) ARGF21
ARCON
SWVON WEV#(100)
SMOVC C00244 BC00244 V=9.2  +MOVJ EC00244
SMOVC C00245 BC00245 V=9.2  +MOVJ EC00245
SMOVC C00246 BC00246 V=9.2  +MOVJ EC00246
SMOVC C00247 BC00247 V=9.2  +MOVJ EC00247
SMOVC C00248 BC00248 V=9.2  +MOVJ EC00248
ARCOF
SFTOF3D
SWVOF
MOVL C00249 BC00249 V=400.0  +MOVJ EC00249 VJ=100.00
MOVL C00250 BC00250 V=1000.0  +MOVJ EC00250 VJ=100.00
MOVJ C00251 BC00251 VJ=100.00  +MOVJ EC00251 VJ=100.00
MOVJ C00252 BC00252 VJ=100.00  +MOVJ EC00252 VJ=100.00
MOVJ C00253 BC00253 VJ=100.00  +MOVJ EC00253 VJ=100.00
'Path W3552
SFTOF3D
SFTON3D P022
MOVJ C00254 BC00254 VJ=100.00  +MOVJ EC00254 VJ=100.00
SMOVL C00255 BC00255 V=333.3  +MOVJ EC00255
SMOVL C00256 BC00256 V=133.3 PL=0  +MOVJ EC00256
SREFP 1 C00257 BC00257  +REFP EC00257
SREFP 2 C00258 BC00258  +REFP EC00258
MACRO1 MJ#(0) ARGF14
ARCON
SMOVC C00259 BC00259 V=8.3  +MOVJ EC00259
SMOVC C00260 BC00260 V=8.3  +MOVJ EC00260
SMOVC C00261 BC00261 V=8.3  +MOVJ EC00261
SMOVC C00262 BC00262 V=8.3  +MOVJ EC00262
SMOVC C00263 BC00263 V=8.3  +MOVJ EC00263
SMOVC C00264 BC00264 V=8.3  +MOVJ EC00264
SMOVL C00265 BC00265 V=8.3  +MOVJ EC00265
ARCOF
SMOVL C00266 BC00266 V=400.0  +MOVJ EC00266
SMOVL C00267 BC00267 V=1000.0  +MOVJ EC00267
SFTOF3D
'Path W3553
SFTOF3D
SFTON3D P022
MOVJ C00268 BC00268 VJ=100.00  +MOVJ EC00268 VJ=100.00
SMOVL C00269 BC00269 V=133.3  +MOVJ EC00269
'SZEROKA SZCZELINA!!!
MACRO1 MJ#(0) ARGF14
SMOVL C00270 BC00270 V=133.3 PL=0  +MOVJ EC00270
SREFP 1 C00271 BC00271  +REFP EC00271
SREFP 2 C00272 BC00272  +REFP EC00272
ARCON
SWVON WEV#(14)
SMOVL C00273 BC00273 V=7.5  +MOVJ EC00273
SMOVL C00274 BC00274 V=7.5  +MOVJ EC00274
ARCOF
SWVOF
SMOVL C00275 BC00275 V=400.0  +MOVJ EC00275
SFTOF3D
SMOVL C00276 BC00276 V=1000.0  +MOVJ EC00276
MOVJ C00277 BC00277 VJ=70.00  +MOVJ EC00277 VJ=70.00
MACRO1 MJ#(0) ARGF14
SFTON3D P088
SMOVL C00278 BC00278 V=166.7  +MOVJ EC00278
ARCON
SMOVL C00279 BC00279 V=10.8  +MOVJ EC00279
ARCOF
SFTOF3D
SMOVL C00280 BC00280 V=250.0  +MOVJ EC00280
'
'NIE SPAWAMY_BRAK BLASZKI
COMM 'Path W3554
COMM SFTOF3D
COMM SFTON3D P023
COMM MOVJ C00281 BC00281 VJ=100.00  +MOVJ EC00281 VJ=100.00
COMM MOVJ C00282 BC00282 VJ=100.00  +MOVJ EC00282 VJ=100.00
COMM SMOVL C00283 BC00283 V=400.0  +MOVJ EC00283
COMM SMOVL C00284 BC00284 V=100.0 PL=0  +MOVJ EC00284
COMM SREFP 1 C00285 BC00285  +REFP EC00285
COMM SREFP 2 C00286 BC00286  +REFP EC00286
COMM MACRO1 MJ#(0) ARGF0
COMM ARCON
COMM SMOVL C00287 BC00287 V=10.0  +MOVJ EC00287
COMM SMOVL C00288 BC00288 V=10.0  +MOVJ EC00288
COMM SMOVL C00289 BC00289 V=10.0  +MOVJ EC00289
COMM ARCOF
COMM SMOVL C00290 BC00290 V=400.0  +MOVJ EC00290
COMM SMOVL C00291 BC00291 V=1000.0  +MOVJ EC00291
COMM SFTOF3D
COMM MOVJ C00292 BC00292 VJ=100.00  +MOVJ EC00292 VJ=100.00
'NIE SPAWAMY_BRAK BLASZKI
COMM 'Path W3555
COMM SFTOF3D
COMM SFTON3D P023
COMM MOVJ C00293 BC00293 VJ=100.00  +MOVJ EC00293 VJ=100.00
COMM SMOVL C00294 BC00294 V=100.0  +MOVJ EC00294
COMM SMOVL C00295 BC00295 V=100.0 PL=0  +MOVJ EC00295
COMM SREFP 1 C00296 BC00296  +REFP EC00296
COMM SREFP 2 C00297 BC00297  +REFP EC00297
COMM MACRO1 MJ#(0) ARGF0
COMM ARCON
COMM SMOVL C00298 BC00298 V=10.0  +MOVJ EC00298
COMM SMOVL C00299 BC00299 V=10.0  +MOVJ EC00299
COMM SMOVL C00300 BC00300 V=10.0  +MOVJ EC00300
COMM ARCOF
COMM SMOVL C00301 BC00301 V=400.0  +MOVJ EC00301
COMM SMOVL C00302 BC00302 V=1000.0  +MOVJ EC00302
COMM SMOVL C00303 BC00303 V=1000.0  +MOVJ EC00303
COMM SFTOF3D
'NIE SPAWAMY_BRAK BLASZKI
COMM 'Path W3556
COMM SFTOF3D
COMM SFTON3D P023
COMM MOVJ C00304 BC00304 VJ=100.00  +MOVJ EC00304 VJ=100.00
COMM SMOVL C00305 BC00305 V=100.0  +MOVJ EC00305
COMM SMOVL C00306 BC00306 V=100.0 PL=0  +MOVJ EC00306
COMM SREFP 1 C00307 BC00307  +REFP EC00307
COMM SREFP 2 C00308 BC00308  +REFP EC00308
COMM MACRO1 MJ#(0) ARGF0
COMM ARCON
COMM SMOVL C00309 BC00309 V=10.0  +MOVJ EC00309
COMM ARCOF
COMM SMOVL C00310 BC00310 V=400.0  +MOVJ EC00310
COMM SMOVL C00311 BC00311 V=1000.0  +MOVJ EC00311
COMM SFTOF3D
'
'NIE SPAWAMY_BRAK BLASZKI
COMM 'Path W3557
COMM SFTOF3D
COMM SFTON3D P024
COMM MOVJ C00312 BC00312 VJ=100.00  +MOVJ EC00312 VJ=100.00
COMM SMOVL C00313 BC00313 V=100.0  +MOVJ EC00313
COMM SMOVL C00314 BC00314 V=100.0 PL=0  +MOVJ EC00314
COMM SREFP 1 C00315 BC00315  +REFP EC00315
COMM SREFP 2 C00316 BC00316  +REFP EC00316
COMM MACRO1 MJ#(0) ARGF0
COMM ARCON
COMM SMOVL C00317 BC00317 V=10.0  +MOVJ EC00317
COMM SMOVL C00318 BC00318 V=10.0  +MOVJ EC00318
COMM SMOVL C00319 BC00319 V=10.0  +MOVJ EC00319
COMM ARCOF
COMM SMOVL C00320 BC00320 V=400.0  +MOVJ EC00320
COMM SMOVL C00321 BC00321 V=1000.0  +MOVJ EC00321
COMM SFTOF3D
COMM MOVJ C00322 BC00322 VJ=100.00  +MOVJ EC00322 VJ=100.00
'NIE SPAWAMY_BRAK BLASZKI
COMM 'Path W3558
COMM SFTOF3D
COMM SFTON3D P024
COMM MOVJ C00323 BC00323 VJ=100.00  +MOVJ EC00323 VJ=100.00
COMM SMOVL C00324 BC00324 V=100.0  +MOVJ EC00324
COMM SMOVL C00325 BC00325 V=100.0 PL=0  +MOVJ EC00325
COMM SREFP 1 C00326 BC00326  +REFP EC00326
COMM SREFP 2 C00327 BC00327  +REFP EC00327
COMM MACRO1 MJ#(0) ARGF0
COMM ARCON
COMM SMOVL C00328 BC00328 V=10.0  +MOVJ EC00328
COMM SMOVL C00329 BC00329 V=10.0  +MOVJ EC00329
COMM SMOVL C00330 BC00330 V=10.0  +MOVJ EC00330
COMM ARCOF
COMM SMOVL C00331 BC00331 V=400.0  +MOVJ EC00331
COMM SMOVL C00332 BC00332 V=1000.0  +MOVJ EC00332
COMM SMOVL C00333 BC00333 V=1000.0  +MOVJ EC00333
COMM SFTOF3D
'NIE SPAWAMY_BRAK BLASZKI
COMM 'Path W3559
COMM SFTOF3D
COMM SFTON3D P024
COMM MOVJ C00334 BC00334 VJ=100.00  +MOVJ EC00334 VJ=100.00
COMM SMOVL C00335 BC00335 V=100.0  +MOVJ EC00335
COMM SMOVL C00336 BC00336 V=100.0 PL=0  +MOVJ EC00336
COMM SREFP 1 C00337 BC00337  +REFP EC00337
COMM SREFP 2 C00338 BC00338  +REFP EC00338
COMM MACRO1 MJ#(0) ARGF0
COMM ARCON
COMM SMOVL C00339 BC00339 V=10.0  +MOVJ EC00339
COMM ARCOF
COMM SMOVL C00340 BC00340 V=400.0  +MOVJ EC00340
COMM SMOVL C00341 BC00341 V=1000.0  +MOVJ EC00341
COMM SFTOF3D
COMM MOVJ C00342 BC00342 VJ=100.00  +MOVJ EC00342 VJ=100.00
'
'NIE SPAWAMY_BRAK BLASZKI
COMM 'Path W3560
COMM SFTOF3D
COMM SFTON3D P025
COMM MOVJ C00343 BC00343 VJ=100.00  +MOVJ EC00343 VJ=100.00
COMM SMOVL C00344 BC00344 V=100.0  +MOVJ EC00344
COMM SMOVL C00345 BC00345 V=100.0 PL=0  +MOVJ EC00345
COMM SREFP 1 C00346 BC00346  +REFP EC00346
COMM SREFP 2 C00347 BC00347  +REFP EC00347
COMM MACRO1 MJ#(0) ARGF0
COMM ARCON
COMM SMOVL C00348 BC00348 V=10.0  +MOVJ EC00348
COMM SMOVL C00349 BC00349 V=10.0  +MOVJ EC00349
COMM SMOVL C00350 BC00350 V=10.0  +MOVJ EC00350
COMM ARCOF
COMM SMOVL C00351 BC00351 V=400.0  +MOVJ EC00351
COMM SMOVL C00352 BC00352 V=1000.0  +MOVJ EC00352
COMM SFTOF3D
COMM MOVJ C00353 BC00353 VJ=100.00  +MOVJ EC00353 VJ=100.00
'NIE SPAWAMY_BRAK BLASZKI
COMM 'Path W3561
COMM SFTOF3D
COMM SFTON3D P025
COMM MOVJ C00354 BC00354 VJ=100.00  +MOVJ EC00354 VJ=100.00
COMM SMOVL C00355 BC00355 V=100.0  +MOVJ EC00355
COMM SMOVL C00356 BC00356 V=100.0 PL=0  +MOVJ EC00356
COMM SREFP 1 C00357 BC00357  +REFP EC00357
COMM SREFP 2 C00358 BC00358  +REFP EC00358
COMM MACRO1 MJ#(0) ARGF0
COMM ARCON
COMM SMOVL C00359 BC00359 V=10.0  +MOVJ EC00359
COMM SMOVL C00360 BC00360 V=10.0  +MOVJ EC00360
COMM SMOVL C00361 BC00361 V=10.0  +MOVJ EC00361
COMM ARCOF
COMM SMOVL C00362 BC00362 V=400.0  +MOVJ EC00362
COMM SMOVL C00363 BC00363 V=1000.0  +MOVJ EC00363
COMM SMOVL C00364 BC00364 V=1000.0  +MOVJ EC00364
COMM SFTOF3D
'NIE SPAWAMY_BRAK BLASZKI
COMM 'Path W3562
COMM SFTOF3D
COMM SFTON3D P025
COMM MOVJ C00365 BC00365 VJ=100.00  +MOVJ EC00365 VJ=100.00
COMM SMOVL C00366 BC00366 V=100.0  +MOVJ EC00366
COMM SMOVL C00367 BC00367 V=100.0 PL=0  +MOVJ EC00367
COMM SREFP 1 C00368 BC00368  +REFP EC00368
COMM SREFP 2 C00369 BC00369  +REFP EC00369
COMM MACRO1 MJ#(0) ARGF0
COMM ARCON
COMM SMOVL C00370 BC00370 V=10.0  +MOVJ EC00370
COMM ARCOF
COMM SMOVL C00371 BC00371 V=400.0  +MOVJ EC00371
COMM SMOVL C00372 BC00372 V=1000.0  +MOVJ EC00372
COMM SFTOF3D
COMM MOVJ C00373 BC00373 VJ=100.00  +MOVJ EC00373 VJ=100.00
COMM MOVJ C00374 BC00374 VJ=100.00  +MOVJ EC00374 VJ=100.00
COMM '
COMM MOVJ C00375 BC00375 VJ=100.00  +MOVJ EC00375 VJ=100.00
COMM MOVJ C00376 BC00376 VJ=100.00  +MOVJ EC00376 VJ=100.00
'NIE SPAWAMY_BRAK BLASZKI
COMM 'Path W3563
COMM SFTOF3D
COMM SFTON3D P023
COMM MOVJ C00377 BC00377 VJ=100.00  +MOVJ EC00377 VJ=100.00
COMM SMOVL C00378 BC00378 V=400.0  +MOVJ EC00378
COMM SMOVL C00379 BC00379 V=100.0 PL=0  +MOVJ EC00379
COMM SREFP 1 C00380 BC00380  +REFP EC00380
COMM SREFP 2 C00381 BC00381  +REFP EC00381
COMM MACRO1 MJ#(0) ARGF0
COMM ARCON
COMM SMOVL C00382 BC00382 V=10.0  +MOVJ EC00382
COMM SMOVL C00383 BC00383 V=10.0  +MOVJ EC00383
COMM SMOVL C00384 BC00384 V=10.0  +MOVJ EC00384
COMM ARCOF
COMM SMOVL C00385 BC00385 V=400.0  +MOVJ EC00385
COMM SMOVL C00386 BC00386 V=1000.0  +MOVJ EC00386
COMM SMOVL C00387 BC00387 V=1000.0  +MOVJ EC00387
COMM SFTOF3D
'NIE SPAWAMY_BRAK BLASZKI
COMM 'Path W3564
COMM SFTOF3D
COMM SFTON3D P023
COMM SMOVL C00388 BC00388 V=100.0  +MOVJ EC00388
COMM SMOVL C00389 BC00389 V=100.0 PL=0  +MOVJ EC00389
COMM SREFP 1 C00390 BC00390  +REFP EC00390
COMM SREFP 2 C00391 BC00391  +REFP EC00391
COMM MACRO1 MJ#(0) ARGF0
COMM ARCON
COMM SMOVL C00392 BC00392 V=10.0  +MOVJ EC00392
COMM SMOVL C00393 BC00393 V=10.0  +MOVJ EC00393
COMM SMOVL C00394 BC00394 V=10.0  +MOVJ EC00394
COMM ARCOF
COMM SMOVL C00395 BC00395 V=400.0  +MOVJ EC00395
COMM SFTOF3D
COMM MOVJ C00396 BC00396 VJ=100.00  +MOVJ EC00396 VJ=100.00
'
COMM MOVJ C00397 BC00397 VJ=100.00  +MOVJ EC00397 VJ=100.00
'NIE SPAWAMY_BRAK BLASZKI
COMM 'Path W3565
COMM SFTOF3D
COMM SFTON3D P024
COMM MOVJ C00398 BC00398 VJ=100.00  +MOVJ EC00398 VJ=100.00
COMM MOVJ C00399 BC00399 VJ=100.00  +MOVJ EC00399 VJ=100.00
COMM SMOVL C00400 BC00400 V=400.0  +MOVJ EC00400
COMM SMOVL C00401 BC00401 V=100.0 PL=0  +MOVJ EC00401
COMM SREFP 1 C00402 BC00402  +REFP EC00402
COMM SREFP 2 C00403 BC00403  +REFP EC00403
COMM MACRO1 MJ#(0) ARGF0
COMM ARCON
COMM SMOVL C00404 BC00404 V=10.0  +MOVJ EC00404
COMM SMOVL C00405 BC00405 V=10.0  +MOVJ EC00405
COMM SMOVL C00406 BC00406 V=10.0  +MOVJ EC00406
COMM ARCOF
COMM SMOVL C00407 BC00407 V=400.0  +MOVJ EC00407
COMM SMOVL C00408 BC00408 V=1000.0  +MOVJ EC00408
COMM SMOVL C00409 BC00409 V=1000.0  +MOVJ EC00409
COMM SFTOF3D
'NIE SPAWAMY_BRAK BLASZKI
COMM 'Path W3566
COMM SFTOF3D
COMM SFTON3D P025
COMM MOVJ C00410 BC00410 VJ=100.00  +MOVJ EC00410 VJ=100.00
COMM SMOVL C00411 BC00411 V=400.0  +MOVJ EC00411
COMM SMOVL C00412 BC00412 V=100.0 PL=0  +MOVJ EC00412
COMM SREFP 1 C00413 BC00413  +REFP EC00413
COMM SREFP 2 C00414 BC00414  +REFP EC00414
COMM MACRO1 MJ#(0) ARGF0
COMM ARCON
COMM SMOVL C00415 BC00415 V=10.0  +MOVJ EC00415
COMM SMOVL C00416 BC00416 V=10.0  +MOVJ EC00416
COMM SMOVL C00417 BC00417 V=10.0  +MOVJ EC00417
COMM ARCOF
COMM SMOVL C00418 BC00418 V=400.0  +MOVJ EC00418
COMM SMOVL C00419 BC00419 V=1000.0  +MOVJ EC00419
COMM SMOVL C00420 BC00420 V=1000.0  +MOVJ EC00420
COMM SFTOF3D
MOVJ C00421 BC00421 VJ=100.00  +MOVJ EC00421 VJ=100.00
MOVJ C00422 BC00422 VJ=100.00  +MOVJ EC00422 VJ=50.00
MOVJ C00423 BC00423 VJ=100.00  +MOVJ EC00423 VJ=50.00
MOVJ C00424 BC00424 VJ=100.00  +MOVJ EC00424 VJ=50.00
MOVJ C00425 BC00425 VJ=100.00  +MOVJ EC00425 VJ=100.00
'Path W3567
SFTOF3D
SFTON3D P021
MOVJ C00426 BC00426 VJ=100.00  +MOVJ EC00426 VJ=100.00
SMOVL C00427 BC00427 V=250.0  +MOVJ EC00427
SMOVL C00428 BC00428 V=133.3 PL=0  +MOVJ EC00428
SREFP 1 C00429 BC00429  +REFP EC00429
SREFP 2 C00430 BC00430  +REFP EC00430
MACRO1 MJ#(0) ARGF21
ARCON
SWVON WEV#(100)
SMOVC C00431 BC00431 V=9.2  +MOVJ EC00431
SMOVC C00432 BC00432 V=9.2  +MOVJ EC00432
SMOVC C00433 BC00433 V=9.2  +MOVJ EC00433
SMOVC C00434 BC00434 V=9.2  +MOVJ EC00434
ARCOF
SWVOF
SMOVL C00435 BC00435 V=400.0  +MOVJ EC00435
SMOVL C00436 BC00436 V=1000.0  +MOVJ EC00436
SFTOF3D
MOVJ C00437 BC00437 VJ=100.00  +MOVJ EC00437 VJ=100.00
'
MOVJ C00438 BC00438 VJ=100.00  +MOVJ EC00438 VJ=100.00
MOVJ C00439 BC00439 VJ=100.00  +MOVJ EC00439 VJ=100.00
'NIE SPAWAMY_BRAK BLASZKI
COMM 'Path W3568
COMM SFTOF3D
COMM SFTON3D P024
COMM MOVJ C00440 BC00440 VJ=100.00  +MOVJ EC00440 VJ=100.00
COMM SMOVL C00441 BC00441 V=100.0  +MOVJ EC00441
COMM SMOVL C00442 BC00442 V=100.0 PL=0  +MOVJ EC00442
COMM SREFP 1 C00443 BC00443  +REFP EC00443
COMM SREFP 2 C00444 BC00444  +REFP EC00444
COMM MACRO1 MJ#(0) ARGF0
COMM ARCON
COMM SMOVL C00445 BC00445 V=10.0  +MOVJ EC00445
COMM SMOVL C00446 BC00446 V=10.0  +MOVJ EC00446
COMM SMOVL C00447 BC00447 V=10.0  +MOVJ EC00447
COMM ARCOF
COMM SMOVL C00448 BC00448 V=400.0  +MOVJ EC00448
COMM SMOVL C00449 BC00449 V=1000.0  +MOVJ EC00449
COMM SFTOF3D
'NIE SPAWAMY_BRAK BLASZKI
COMM 'Path W3569
COMM SFTOF3D
COMM SFTON3D P025
COMM MOVJ C00450 BC00450 VJ=100.00  +MOVJ EC00450 VJ=100.00
COMM SMOVL C00451 BC00451 V=100.0  +MOVJ EC00451
COMM SMOVL C00452 BC00452 V=100.0 PL=0  +MOVJ EC00452
COMM SREFP 1 C00453 BC00453  +REFP EC00453
COMM SREFP 2 C00454 BC00454  +REFP EC00454
COMM MACRO1 MJ#(0) ARGF0
COMM ARCON
COMM SMOVL C00455 BC00455 V=10.0  +MOVJ EC00455
COMM SMOVL C00456 BC00456 V=10.0  +MOVJ EC00456
COMM SMOVL C00457 BC00457 V=10.0  +MOVJ EC00457
COMM ARCOF
COMM SMOVL C00458 BC00458 V=400.0  +MOVJ EC00458
COMM SMOVL C00459 BC00459 V=1000.0  +MOVJ EC00459
COMM SMOVL C00460 BC00460 V=1000.0  +MOVJ EC00460
COMM SFTOF3D
COMM MOVJ C00461 BC00461 VJ=100.00  +MOVJ EC00461 VJ=100.00
COMM '
COMM MOVJ C00462 BC00462 VJ=100.00  +MOVJ EC00462 VJ=100.00
COMM MOVJ C00463 BC00463 VJ=100.00  +MOVJ EC00463 VJ=100.00
'Path W3570
SFTOF3D
SFTON3D P026
MOVJ C00464 BC00464 VJ=100.00  +MOVJ EC00464 VJ=100.00
MOVJ C00465 BC00465 VJ=100.00  +MOVJ EC00465 VJ=100.00
SMOVL C00466 BC00466 V=666.7  +MOVJ EC00466
SMOVL C00467 BC00467 V=133.3  +MOVJ EC00467
SREFP 1 C00468 BC00468  +REFP EC00468
SREFP 2 C00469 BC00469  +REFP EC00469
MACRO1 MJ#(0) ARGF21
ARCON
SMOVL C00470 BC00470 V=7.5  +MOVJ EC00470
SMOVL C00471 BC00471 V=7.5  +MOVJ EC00471
SMOVL C00472 BC00472 V=7.5  +MOVJ EC00472
SMOVL C00473 BC00473 V=7.5  +MOVJ EC00473
SMOVL C00474 BC00474 V=7.5  +MOVJ EC00474
SMOVL C00475 BC00475 V=7.5  +MOVJ EC00475
SMOVL C00476 BC00476 V=7.5  +MOVJ EC00476
ARCON
SMOVL C00477 BC00477 V=7.5  +MOVJ EC00477
SMOVL C00478 BC00478 V=7.5  +MOVJ EC00478
SMOVL C00479 BC00479 V=7.5  +MOVJ EC00479
SMOVL C00480 BC00480 V=7.5  +MOVJ EC00480
ARCOF
SMOVL C00481 BC00481 V=250.0  +MOVJ EC00481
SMOVL C00482 BC00482 V=1000.0  +MOVJ EC00482
SFTOF3D
MOVJ C00483 BC00483 VJ=100.00  +MOVJ EC00483 VJ=100.00
'jakie searche do takicj spoin?
MOVJ C00484 BC00484 VJ=100.00  +MOVJ EC00484 VJ=100.00
MOVJ C00485 BC00485 VJ=100.00  +MOVJ EC00485 VJ=100.00
'Path W3572
SFTOF3D
'jakie searche do takicj spoin?
MOVJ C00486 BC00486 VJ=100.00  +MOVJ EC00486 VJ=100.00
'Path W3579
SFTOF3D
MOVJ C00487 BC00487 VJ=50.00  +MOVJ EC00487 VJ=100.00
COMM PAUSE
COMM MOVL C00488 BC00488 V=400.0  +MOVJ EC00488 VJ=100.00
COMM SFTOF3D
COMM SFTON3D P089
COMM SMOVL C00489 BC00489 V=100.0 PL=0  +MOVJ EC00489
COMM SREFP 1 C00490 BC00490  +REFP EC00490
COMM SREFP 2 C00491 BC00491  +REFP EC00491
COMM MACRO1 MJ#(0) ARGF9
COMM ARCON
COMM SMOVL C00492 BC00492 V=11.7  +MOVJ EC00492
COMM ARCOF
COMM MOVL C00493 BC00493 V=666.7  +MOVJ EC00493 VJ=100.00
COMM SMOVL C00494 BC00494 V=166.7  +MOVJ EC00494
COMM ARCON
COMM SMOVL C00495 BC00495 V=11.7  +MOVJ EC00495
COMM ARCOF
COMM SFTOF3D
SMOVL C00496 BC00496 V=250.0  +MOVJ EC00496
MACRO1 MJ#(0) ARGF14
MOVL C00497 BC00497 V=1000.0  +MOVJ EC00497 VJ=100.00
SFTON3D P090
SMOVL C00498 BC00498 V=166.7  +MOVJ EC00498
ARCON
SMOVL C00499 BC00499 V=12.5  +MOVJ EC00499
ARCOF
SMOVL C00500 BC00500 V=166.7  +MOVJ EC00500
SMOVL C00501 BC00501 V=166.7  +MOVJ EC00501
SMOVL C00502 BC00502 V=166.7  +MOVJ EC00502
ARCON
SMOVL C00503 BC00503 V=10.8  +MOVJ EC00503
ARCOF
SMOVL C00504 BC00504 V=166.7  +MOVJ EC00504
SFTOF3D
SMOVL C00505 BC00505 V=1000.0  +MOVJ EC00505
MOVJ C00506 BC00506 VJ=100.00  +MOVJ EC00506 VJ=100.00
COMM MOVJ C00507 BC00507 VJ=100.00  +MOVJ EC00507 VJ=100.00
COMM MOVJ C00508 BC00508 VJ=100.00  +MOVJ EC00508 VJ=100.00
'NIE SPAWAMY
COMM 'Path W3582
COMM SFTOF3D
COMM PAUSE
COMM SFTON3D P031
COMM MOVJ C00509 BC00509 VJ=100.00  +MOVJ EC00509 VJ=100.00
COMM SMOVL C00510 BC00510 V=100.0  +MOVJ EC00510
COMM SMOVL C00511 BC00511 V=100.0 PL=0  +MOVJ EC00511
COMM SREFP 1 C00512 BC00512  +REFP EC00512
COMM SREFP 2 C00513 BC00513  +REFP EC00513
COMM MACRO1 MJ#(0) ARGF0
COMM ARCON
COMM SMOVL C00514 BC00514 V=10.0  +MOVJ EC00514
COMM SMOVL C00515 BC00515 V=10.0  +MOVJ EC00515
COMM SMOVL C00516 BC00516 V=10.0  +MOVJ EC00516
COMM ARCOF
COMM SMOVL C00517 BC00517 V=400.0  +MOVJ EC00517
COMM SMOVL C00518 BC00518 V=1000.0  +MOVJ EC00518
COMM SFTOF3D
'Down
MOVJ C00519 BC00519 VJ=100.00  +MOVJ EC00519 VJ=100.00
END
